VAR 
MesDataExd				: Datalogger_SENECA;                		
	
//INPUT Modbus
	FB_ModbusRead	          	: ARRAY[1..2] OF FB_ModbusRead; 	            // (NA) FB for Modbus Reading	
	MesBlock1_Temp				: ARRAY [1..8] OF WORD ; 
	
	AlarmModbusInput			: BOOL;
	AlarmID_ModbusInput			: UDINT;
END_VAR

METHOD M_AlarmManagement
//////////////////
// Generates object alarms and manages resets 
//////////////////

VAR 
	// Method local variables (reinitialized at each cycle) 
	FB_AlarmCodeManager		: FB_AlarmCodeManager;  
	Transfo_Synthesis		: INT;
END_VAR
	
// ALARM CODE //
	FB_AlarmCodeManager(
		bAlarm1				:= FALSE,														// 
		bAlarm2				:= FALSE,														// 
		bAlarm3				:= FALSE,														// 
		bAlarm4				:= FALSE,														//
		bAlarm5				:= FALSE,														//
		bAlarm6				:= FALSE,														//
		bAlarm7				:= FALSE,														//
		bAlarm8				:= FALSE,														//
		bAlarm9				:= FALSE,														//
		bAlarm10			:= FALSE,														//
		bAlarm11			:= FALSE, 														// 
		bAlarm12			:= FALSE, 														// 
		bAlarm13			:= FALSE, 														//                                          
		bAlarm14			:= FALSE,														//                                          
		bAlarm15			:= FALSE,														// 		
		wAlarmCode			=>MesDataExd.MesData.MesAlarmCode);										//
			
// WARNING CODE //
	FB_AlarmCodeManager(
		bAlarm1				:= AlarmModbusInput, 											// Error Modbus read of the datalogger data
		bAlarm2				:= FALSE, 														//
		bAlarm3				:= FALSE,														//
		bAlarm4				:= FALSE,														//
		bAlarm5				:= FALSE,														//
		bAlarm6				:= FALSE,														//
		bAlarm7				:= FALSE,														//
		bAlarm8				:= FALSE,														//
		bAlarm9				:= FALSE,														//
		bAlarm10			:= FALSE,														//
		bAlarm11			:= FALSE,														//
		bAlarm12			:= FALSE,														//
		bAlarm13			:= FALSE,														//
		bAlarm14			:= FALSE,														//
		bAlarm15			:= FALSE,														//
		wAlarmCode			=>MesDataExd.MesData.MesWarningCode);										//
		                                                        							
// EVENT CODE //                                                							                                                     							
	FB_AlarmCodeManager(                                        							
		bAlarm1				:= FALSE,						    							//  
		bAlarm2				:= FALSE, 														//  
		bAlarm3				:= FALSE,														//
		bAlarm4				:= FALSE,														//
		bAlarm5				:= FALSE,														//
		bAlarm6				:= FALSE,														//
		bAlarm7				:= FALSE,														//
		bAlarm8				:= FALSE,														//
		bAlarm9				:= FALSE,														//
		bAlarm10			:= FALSE,														//
		bAlarm11			:= FALSE,														//
		bAlarm12			:= FALSE,														//
		bAlarm13			:= FALSE,														//
		bAlarm14			:= FALSE,														//
		bAlarm15			:= FALSE,														//
		wAlarmCode			=>MesDataExd.MesData.MesEventCode);										//
		
MesDataExdMesDataExd		:= MesDataExd.MesData.
END_METHOD

METHOD M_CP

VAR 
	// Method local variables (reinitialized at each cycle) 
	
END_VAR

Trig_Cmd_Read(CLK:=IN_CmdToggleRead);

IF Trig_Cmd_Read.Q THEN
	IN_CmdToggleRead := FALSE;
	MesCP_Read := NOT MesCP_Read;
END_IF
END_METHOD

METHOD M_Execute : BOOL
VAR_INPUT
END_VAR
IF bInit THEN
	M_Init();
	bInit := FALSE;
ELSIF CmdInit_G THEN 
	bInit:= TRUE ;
END_IF

SUPER^.M_Execute() ;
END_METHOD

METHOD M_Init : BOOL
VAR_INPUT
END_VAR
END_METHOD


METHOD M_Read : BOOL
VAR_INPUT
END_VAR

VAR
	MW					: FB_MergeWordsToFloat;
END_VAR
// CP-Read / Write 

MesDataExd.MesData.MesCP_Read := MesCP_Read ; 
MesDataExd.MesData.MesCP_Write := MesCP_Write ;  

IF MesCP_Read  THEN	
// MODBUS Read	
	FB_ModbusRead[1]
		(
			nTCPPort		:= ParamTcpPort,
			ClockRead		:= MesCP_Read AND ClockRead, 
			Reset			:= CmdClearFault_G OR IN_CmdReset_L,
			sIPAddr			:= ParamIPAddress ,
			nUnitID			:= 1, 
			tTimeout		:= ParamWriteTimeout,
			nQuantity		:= 4, 
			nMBAddr			:= 40005, 
			cbLength		:= SIZEOF(MesBlock1_Temp), 
			pDestAddr		:= ADR(MesBlock1_Temp), 
			ModbusReadAlarm	=> AlarmModbusInput, 
			ErrorId			=> AlarmID_ModbusInput
		);
	
// Wind Data : Float AB CD	
	MW( WORD_STRONG:= MesBlock1_Temp[1  ],	WORD_WEAK := MesBlock1_Temp[2  ], VAR_OUT := MesDataExd.MesData.MesWindSp);		
	MW( WORD_STRONG:= MesBlock1_Temp[3  ],	WORD_WEAK := MesBlock1_Temp[4  ], VAR_OUT := MesDataExd.MesData.MesWindDir);
END_IF
END_METHOD

METHOD M_Write : BOOL
VAR
		
		
END_VAR
END_METHOD

END_FUNCTION_BLOCK

// ---- 01_Equipement_Library/GRID/FB_GRID_Base.TcPOU
FUNCTION_BLOCK FB_GRID_Base 
//////////////////
// Grid Operator interface. Base FB.
//////////////////
VAR_INPUT PERSISTENT
	// Parameters of the Object (instance specific) 
	
END_VAR

VAR_INPUT
	// I/O Inputs 
		MesConnectOrderIO			: BOOL ; 					// (NA) 
		MesDisconnectOrderIO 		: BOOL ; 					// (NA) 	
		
END_VAR

VAR_OUTPUT
	//Child objects
	
END_VAR
VAR
	//M_ALARMMANAGEMENT VARIABLES//                                                    								
//	MesDataExd				: GRID ;                   								
		
	//M_INIT VARIABLES //
		bInit						: BOOL:= TRUE ; 			// (NA) Initialize object parameters at first cycle 
		
	// M_EXECUTE VARIABLES //
	
   		MesCP_Read					: BOOL := TRUE;	(* Read function enable *)
		

                      	
END_VAR

METHOD M_AlarmManagement
//////////////////
// Digiware measurement tool alarm and warning management
/////////////////

VAR 
	
END_VAR
END_METHOD

METHOD M_CP

VAR 
	// Method local variables (reinitialized at each cycle) 
	
END_VAR
END_METHOD

METHOD M_Evaluate
//////////////////
//  Read Modbus Variable for PCS. 
/////////////////
VAR 
	// Method local variables (reinitialized at each cycle) 
	
END_VAR
END_METHOD

METHOD M_Execute
//////////////////
//  Method Calls 
/////////////////
VAR 
	// Method local variables (reinitialized at each cycle) 

END_VAR

// PERMANENT CONDITIONS //
	M_CP() ; 
	
// METHODS CALLS //
	IF bInit THEN
		M_Init() ; 
		bInit					:= FALSE ; 
	ELSIF CmdInit_G THEN 
		bInit:= TRUE ;
		
	END_IF

	M_Evaluate() ; 
	M_AlarmManagement();
END_METHOD

METHOD M_Init
VAR 

END_VAR
END_METHOD

END_FUNCTION_BLOCK

// ---- 01_Equipement_Library/GRID/FB_GRID_Enedis.TcPOU
FUNCTION_BLOCK FB_GRID_Enedis EXTENDS FB_GRID_Base
//////////////////
// Grid Operator interface. Base FB
//////////////////
VAR_INPUT PERSISTENT
	// Parameters of the Object (instance specific) 
		{attribute 'OPC.UA.DA' := '1'} 
		ParamRseAvailable						: BOOL:=TRUE;		(* (NA) GRID with RSE option*)
		{attribute 'OPC.UA.DA' := '1'} 
		ParamTaAvailable						: BOOL:=TRUE;		(* (NA) GRID with Teleaction option*)
		{attribute 'OPC.UA.DA' := '1'} 
		ParamP0Available						: BOOL:=TRUE; 		(* (NA) GRID with P regulation option*)
		{attribute 'OPC.UA.DA' := '1'} 
		ParamQ0Available						: BOOL:=TRUE; 		(* (NA) GRID with Q regulation option*)
		ParamTONFiltering						: TIME:=T#200MS; 	(* (ms) Minimum tempo filter before command validation (noise filtering)*)
		{attribute 'OPC.UA.DA' := '1'} 
		ParamPmaxPark							: REAL;				(* (kW) Contractual maximal power plant active power*)
		{attribute 'OPC.UA.DA' := '1'} 
		ParamQMax								: REAL;				(* (Kvar) Contractual maximal power plant reactive power*)
		{attribute 'OPC.UA.DA' := '1'} 
		ParamQMin								: REAL; 			(* (Kvar) Contractual maximal power plant reactive power*)
		{attribute 'OPC.UA.DA' := '1'} 
		ParamPMin								: REAL;				(* (kW)   Contractual minimal power plant active power*)
		
		MesDataExd								: GRID_Enedis;
END_VAR


VAR_INPUT
	// I/O Inputs 
		//FROM ENEDIS
		IN_CmdAutCpl_IO							: BOOL; 			//Coupling Authorization (Autorisation de couplage				)
		IN_CmdDisconnect_End_IO					: BOOL; 			//End of disconnect order(Fin de demande de decouplage         )
		IN_CmdDisconnect_IO						: BOOL;				//Disconnect order(Demande de decouplage                )
		IN_CmdRSEOn_IO							: BOOL;				//Start of RSE (Mise en RSE                          )
		IN_CmdRSEOff_IO							: BOOL;				//Stop of RSE (Mise Hors RSE                        )
		IN_CmdTAOn_IO							: BOOL; 			//Teleaction in service(Teleaction en service                )
		IN_CmdTAOff_IO							: BOOL; 			//Teleaction out of service (Teleaction Hors service              )
		IN_CmdStopPReg_IO						: BOOL;				//Desactivation of P0 regulation(Fin de passage a P0                  )
		IN_CmdStartPReg_IO						: BOOL;				//Activation of P0 regulation (Passage a P0                         )
		IN_CmdStopQReg_IO						: BOOL;				//Desactivation of Q0 regulation(Fin de passage a Q0                  )
		IN_CmdStartQreg_IO						: BOOL;				//Activation of Q0 regulation(Passage a Q0                         )
		IN_CmdEmergencyDisconnect_End_IO		: BOOL;				// End of Emergency disconnect order(Fin demande d'effacement d'urgence	)	
		IN_CmdEmergencyDisconnect_IO			: BOOL;				// Emergency disconnect order(Demande d'effacement d'urgence       )
		IN_CmdDisconnectFromTac_IO				: BOOL; 			// Teleaction disconnect(Decouplage par tac                   )
		IN_CmdTacInFault_IO						: BOOL; 			//Teleaction in fault(Défaut Tac							)
		IN_CmdSynchro_IO						: BOOL;				// Syncrhonization signal
		(* 4..20mA *)                                   			
		IN_MesP0Reg_IO							: INT; 				// (kW) Grid P0
		IN_MesQ0Reg_IO							: INT; 				// (Kvar) Grid Q0
		                                                			
		                                                			
		//FROM AKSES                                    			
		IN_CmdAutCpl_other						: BOOL; 			
		IN_CmdEmergencyDisconnect_other			: BOOL; 			
		IN_CmdEmergencyDisconnect_End_other		: BOOL; 			
		IN_CmdDisconnect_other					: BOOL; 			
		IN_CmdDisconnect_end_other				: BOOL; 			
		IN_CmdStartPReg_other					: BOOL; 			
		IN_CmdStartQReg_other					: BOOL; 			
		IN_CmdStopPReg_other					: BOOL; 			
		IN_CmdStopQReg_other					: BOOL; 			
		                                                			
		(*TC Relais Protection*)                        			
		IN_ConnectAuthorizationLost				: BOOL; 			// Tous les cas pour un Reset aut Couplage recu
		IN_Unavailable							: BOOL; 			// Disjoncteur général en Local, ou tous les départs en Local ou Bouton d'arret d'urgence 
		IN_PP_Connected							: BOOL; 			// Centrale Couplée si DG = Fermé et au moins 1 départ antenne en production et au moins un onduleur en Prod
                                                        			
END_VAR                                                 			
                                                        			
                                                        			
VAR_OUTPUT                                              			
		OUT_MesPPUnavailable_IO					: BOOL; 			// TS centrale indisponible
		OUT_MesPPConnected_IO					: BOOL; 			// Centrale couplée(1)/Centrale Découplée(0)
		OUT_MesPPDisconnected_IO				: BOOL; 			(*Centrale Découplée*)
		OUT_MesAutCpl_IO 						: BOOL; 			// Autorisation de couplage reçue(1)/Attente d'autorisation de couplage(0)
		OUT_MesAutCpl_end_IO 					: BOOL; 			(*Autorisation de couplage attente*)
		OUT_MesDisconnect_IO 					: BOOL; 			// Demande de découplage reçue(1)/Fin de demande de découplage(0)
		OUT_MesDisconnect_End_IO 				: BOOL; 			(*Demande de découplage attente*)
		OUT_MesEmergencyDisconnect_IO 			: BOOL; 			// Demande d effacement d'urgence reçue
		OUT_MesEmergencyDisconnect_End_IO 		: BOOL; 			(*Demande d effacement d'urgence attente*)		
		OUT_MesRSEON_IO							: BOOL; 			// Demande mise en RSE reçue
		OUT_MesRSEOff_IO						: BOOL; 			// Demande mise en RSE en attente
		OUT_MesTAOn_IO							: BOOL; 			// Demande mise en TeleAction reçue
		OUT_MesTAOff_IO							: BOOL; 			// Demande mise en TeleAction en attente
		OUT_MesStartPReg_IO						: BOOL; 			// Demande mise en regulation de P reçue
		OUT_MesStopPReg_IO						: BOOL; 			// Demande mise en regulation de P en attente
		OUT_MesStartQReg_IO						: BOOL; 			// Demande mise en regulation de Q reçue
		OUT_MesStopQReg_IO						: BOOL; 			// Demande mise en regulation de Q en attente	
END_VAR

VAR
		//TON
		TONConnectAuthorization					: TON;
		TONEmergencyDisconnect	               	: TON;
	    TONEmergencyDisconnect_end	            : TON;
	    TONDisconnect	                		: TON;
	    TONDisconnect_end                		: TON;
	    TONPRegOn				                : TON;
	    TONPRegOff				                : TON;
	    TONQregOn				                : TON;
	    TONQRegOff				                : TON;
	    TONRSEOn				                : TON;
	    TONRSEOff				                : TON;
	    TONTAOn					                : TON;
	    TONTAOff				                : TON;
				
END_VAR

METHOD M_AlarmManagement
//////////////////
// alarm and warning management
/////////////////

VAR 
	FB_AlarmCodeManager			: FB_AlarmCodeManager ; 
	
END_VAR
// ALARM CODE //
	FB_AlarmCodeManager(
		bAlarm1			:=MesDataExd.MesData.OUT_MesPPUnavailable, // Power plant is unavailable
		bAlarm2			:=FALSE, //
		bAlarm3			:=FALSE, //
		bAlarm4			:=FALSE, //
		bAlarm5			:=FALSE, //
		bAlarm6			:=FALSE, //
		bAlarm7			:=FALSE, //
		bAlarm8			:=FALSE, //
		bAlarm9			:=FALSE, //
		bAlarm10		:=FALSE, //
		bAlarm11		:=FALSE, //
		bAlarm12		:=FALSE, //
		bAlarm13		:=FALSE, //
		bAlarm14		:=FALSE, //
		bAlarm15		:=FALSE, //						 
		wAlarmCode		=>MesDataExd.MesData.MesAlarmCode);

// WARNING CODE //
	FB_AlarmCodeManager(		
		bAlarm1			:=IN_ConnectAuthorizationLost, 							//Loss of coupliong authorization
		bAlarm2			:=FALSE,													//			
		bAlarm3			:=MesDataExd.MesData.OUT_SetptP > ParamPmaxPark OR MesDataExd.MesData.OUT_SetptP <= 0 ,		// P Setpoint from grid outside of permitted range
		bAlarm4			:=MesDataExd.MesData.OUT_SetptQ > ParamQMax OR MesDataExd.MesData.OUT_SetptQ <= ParamQMin, 	// Q Setpoint from grid outside of permitted range
		bAlarm5			:=MesDataExd.MesData.OUT_MesPPConnected						, 	//Powerplant is connected  
		bAlarm6			:=NOT MesDataExd.MesData.OUT_MesPPConnected					, 	//Powerplant is disconnected
		bAlarm7			:=MesDataExd.OUT_CmdPReg							    , 	//Q regulation mode is active     
		bAlarm8			:=NOT MesDataExd.MesData.OUT_CmdAutCpl		    		, 	//Waiting for coupling authorization	
		bAlarm9			:=MesDataExd.MesData.OUT_CmdDisconnect				, 	//Disconnect order
		bAlarm10		:=MesDataExd.MesData.OUT_CmdEmergencyDisconnect 	        , 	//Emergency Disconnect order
		bAlarm11		:=MesDataExd.OUT_CmdPReg												, 	// P regulation mode is active
		bAlarm12		:=MesDataExd.OUT_Rse								    , 	// RSE mode active  
		bAlarm13		:=MesDataExd.OUT_TA 							, 	//Teleaction active
		bAlarm14		:=IN_CmdDisconnectFromTac_IO , 		// Disconnect order from TAC
		bAlarm15		:=IN_CmdTacInFault_IO , 			// TAC in Fault 
		wAlarmCode		=>MesDataExd.MesData.MesWarningCode);		

// EVENT CODE 1//
	FB_AlarmCodeManager(
		bAlarm1			:=FALSE , // 
		bAlarm2			:=NOT MesDataExd.OUT_CmdPReg							    , 	//P regulation mode is inactive
		bAlarm3			:=MesDataExd.MesData.OUT_CmdAutCpl					, 	//Coupling authorization
		bAlarm4			:=FALSE ,//
		bAlarm5			:=IN_CmdSynchro_IO			    						, 	// Synchronization signal 
		bAlarm6			:=NOT MesDataExd.MesData.OUT_CmdDisconnect			, 	//End of disconnect order 
		bAlarm7			:=MesDataExd.MesData.OUT_CmdDisconnect				, 	//Disconnect order
		bAlarm8			:=NOT MesDataExd.MesData.OUT_CmdEmergencyDisconnect					, 	//End of Emergency Disconnect order
		bAlarm9			:=MesDataExd.MesData.OUT_CmdEmergencyDisconnect 	        , 	//Emergency Disconnect order
		bAlarm10		:=MesDataExd.OUT_CmdPReg												, 	// P regulation mode is active
		bAlarm11		:=NOT MesDataExd.OUT_CmdPReg												, 	//P regulation mode is inactive
		bAlarm12		:=MesDataExd.OUT_Rse								    , 	// RSE mode active    
		bAlarm13		:=NOT MesDataExd.OUT_Rse							    , 	//RSE mode inactive  
		bAlarm14		:=MesDataExd.OUT_TA 							, 	//Teleaction active
		bAlarm15		:=NOT MesDataExd.OUT_TA							, 	//Teleaction inactive
		wAlarmCode		=>MesDataExd.MesData.MesEventCode);   
                          	
// EVENT CODE 2 //		                                              	
	FB_AlarmCodeManager(                                              	
		bAlarm1			:=IN_CmdAutCpl_IO , 							// Autorisation de couplage du DEIE
		bAlarm2			:=IN_CmdDisconnect_End_IO,						// Fin de demande de découplage du DEIE
		bAlarm3			:=IN_CmdDisconnect_IO		   , 				// Demande de decouplage du DEIE
		bAlarm4			:= IN_CmdEmergencyDisconnect_End_IO	   	, 		// Emergency disconnect
		bAlarm5			:=IN_CmdAutCpl_other, 							// Autorisation de couplage du DEIE de la HMI
		bAlarm6			:=IN_CmdDisconnect_other		 , 				// Demande de decouplage du DEIE de la HMI
		bAlarm7			:=IN_CmdDisconnect_end_other,	 				// Demande de decouplage par TAC de la HMI
		bAlarm8			:=FALSE	, 										// 
		bAlarm9			:=IN_Unavailable, 								// Centrale indisponible dans le code
		bAlarm10		:=FALSE, 	//
		bAlarm11		:=FALSE	, 	//
		bAlarm12		:=FALSE, 	//
		bAlarm13		:=FALSE, 	//       
		bAlarm14		:=FALSE, 	//
		bAlarm15		:=FALSE	,//
		wAlarmCode		=>MesDataExd.MesData.MesEventCode2);
END_METHOD

METHOD M_CP
//////////////////
//  Emulator
/////////////////

VAR 
	// Method local variables (reinitialized at each cycle) 
	
END_VAR
END_METHOD

METHOD M_Evaluate
//////////////////
//  Evaluate grid variables 
/////////////////
VAR 
	// Method local variables (reinitialized at each cycle) 
	WatchDog	: BOOL;
END_VAR
WatchDog		:= TRUE;

//Filtering Input
	TONConnectAuthorization		(IN:=IN_CmdAutCpl_IO,PT:=ParamTONFiltering);
	TONEmergencyDisconnect		(IN:=IN_CmdEmergencyDisconnect_IO,PT:=ParamTONFiltering);	
	TONEmergencyDisconnect_end	(IN:=IN_CmdEmergencyDisconnect_End_IO,PT:=ParamTONFiltering);	
	TONDisconnect				(IN:=IN_CmdDisconnect_IO,PT:=ParamTONFiltering);	
	TONDisconnect_end			(IN:=IN_CmdDisconnect_End_IO,PT:=ParamTONFiltering);
	TONPRegOn				(IN:=IN_CmdStartPReg_IO,PT:=ParamTONFiltering);			
	TONPRegOff				(IN:=IN_CmdStopPReg_IO,PT:=ParamTONFiltering);				
	TONQregOn				(IN:=IN_CmdStartQreg_IO,PT:=ParamTONFiltering);				
	TONQRegOff				(IN:=IN_CmdStopQReg_IO,PT:=ParamTONFiltering);				
	TONRSEOn				(IN:=IN_CmdRSEOn_IO,PT:=ParamTONFiltering);				
	TONRSEOff				(IN:=IN_CmdRSEOff_IO,PT:=ParamTONFiltering);				
	TONTAOn					(IN:=IN_CmdTAOn_IO,PT:=ParamTONFiltering);					
	TONTAOff				(IN:=IN_CmdTAOff_IO,PT:=ParamTONFiltering);		

//Converting P0 & Q0
	IF ParamP0Available THEN
		//OUT_P0 :=  (MesP0RegIO/ 32767.0) * REAL_TO_INT(ParamPmaxPark);
	MesDataExd.MesData.OUT_SetptP :=  (IN_MesP0Reg_IO/ 32767.0) * ABS(ParamPMin - ParamPmaxPark) + (ParamPMin);
	END_IF
	IF ParamQ0Available THEN
	MesDataExd.MesData.OUT_SetptQ := ( IN_MesQ0Reg_IO / 32767.0) * ABS(ParamQMin - ParamQMax) + (ParamQMin);
	END_IF	
//Logical Equation
	(*PLCUnavailable Si Watchdog n'est pas mis a jour a chaque temps de cycle Ou que la centrale est en Local *)
	MesDataExd.MesData.OUT_MesPPUnavailable := NOT WatchDog OR IN_Unavailable;
	
	(*Centrale Couplée *)
	MesDataExd.MesData.OUT_MesPPConnected := IN_PP_Connected;
	
	(*Autorisation de couplage*)
		IF TONConnectAuthorization.Q OR IN_CmdAutCpl_other THEN
		MesDataExd.MesData.OUT_CmdAutCpl := 1 ;
		END_IF
		
	(*Défaut GTE > 50s : Reset Aut Couplage recus*)
	(*Défaut C13_100 : Reset Aut Couplage recus*)
		IF IN_ConnectAuthorizationLost THEN  //IN_Long_GTE_Fault OR IN_C13_100_Fault OR IN_UnknownFault OR IN_3GTE_Fault THEN
		MesDataExd.MesData.OUT_CmdAutCpl  := FALSE ;
		END_IF
	
	(* RESEAU 6 ET 7 - DEMANDE DE DECOUPLAGE*)
		IF TONDisconnect.Q OR IN_CmdDisconnect_other THEN
			MesDataExd.MesData.OUT_CmdDisconnect := 1 ;
		END_IF
	
		IF TONDisconnect_end.Q OR IN_CmdDisconnect_end_other THEN
		MesDataExd.MesData.OUT_CmdDisconnect := 0 ;
		END_IF

	(* RESEAU 8 ET 9 - DEMANDE D’EFFACEMENT D’URGENCE*)
		IF TONEmergencyDisconnect.Q OR  IN_CmdEmergencyDisconnect_other THEN
		MesDataExd.MesData.OUT_CmdEmergencyDisconnect := 1 ;
		END_IF
	
		IF TONEmergencyDisconnect_end.Q OR IN_CmdEmergencyDisconnect_End_other THEN
		MesDataExd.MesData.OUT_CmdEmergencyDisconnect := 0 ;
		END_IF
	(* RESEAU 10 ET 11 - PASSAGE A P0*)
		IF TONPRegOn.Q OR IN_CmdStartPReg_other THEN
		MesDataExd.OUT_CmdPReg := 1 ;
		END_IF
		
		IF TONPRegOff.Q OR IN_CmdStopPReg_other THEN
		MesDataExd.OUT_CmdPReg := 0 ;
		END_IF
		
	(* RESEAU 12 ET 13 - PASSAGE A Q0*)
		IF TONQregOn.Q OR IN_CmdStartQReg_other THEN
		MesDataExd.OUT_CmdQReg := 1 ;
		END_IF
		
		IF TONQregOff.Q OR IN_CmdStopQReg_other THEN
		MesDataExd.OUT_CmdQReg := 0 ;
		END_IF

				
	(* RSE*)
		IF TONRSEOn.Q  THEN
		MesDataExd.OUT_Rse := 1 ;
		ELSIF TONRSEOff.Q THEN
		MesDataExd.OUT_Rse := 0 ;
		END_IF
		
	(* TA*)
		IF TONTAOn.Q  THEN
		MesDataExd.OUT_TA := 1 ;
		ELSIF TONTAOff.Q THEN
		MesDataExd.OUT_TA := 0 ;
		END_IF
		
	
// Update Outputs IO to GRID 
OUT_MesPPUnavailable_IO				:= MesDataExd.MesData.OUT_MesPPUnavailable ; 			
OUT_MesPPConnected_IO				:= MesDataExd.MesData.OUT_MesPPConnected ; 	
OUT_MesPPDisconnected_IO			:= NOT MesDataExd.MesData.OUT_MesPPConnected ; 
OUT_MesAutCpl_IO 					:= MesDataExd.MesData.OUT_CmdAutCpl ; 			
OUT_MesAutCpl_end_IO 				:= NOT MesDataExd.MesData.OUT_CmdAutCpl ; 		
OUT_MesDisconnect_IO 				:= MesDataExd.MesData.OUT_CmdDisconnect ; 		
OUT_MesDisconnect_End_IO 			:= NOT MesDataExd.MesData.OUT_CmdDisconnect ; 		
OUT_MesEmergencyDisconnect_IO 		:= MesDataExd.MesData.OUT_CmdEmergencyDisconnect ; 		
OUT_MesEmergencyDisconnect_End_IO 	:= NOT MesDataExd.MesData.OUT_CmdEmergencyDisconnect ; 		

OUT_MesRSEON_IO						:= MesDataExd.OUT_Rse ;
OUT_MesRSEOff_IO					:= NOT MesDataExd.OUT_Rse ;
OUT_MesTAOn_IO						:= MesDataExd.OUT_TA ; 
OUT_MesTAOff_IO						:= NOT MesDataExd.OUT_TA ; 

OUT_MesStartPReg_IO	 := MesDataExd.OUT_CmdPReg ; 
OUT_MesStopPReg_IO	 := NOT MesDataExd.OUT_CmdPReg ; 
OUT_MesStartQReg_IO	 := MesDataExd.OUT_CmdQReg ; 
OUT_MesStopQReg_IO	 := NOT MesDataExd.OUT_CmdQReg ;
END_METHOD

METHOD M_Execute
//////////////////
//  Method Calls 
/////////////////
VAR 
	// Method local variables (reinitialized at each cycle) 
	
END_VAR
// PERMANENT CONDITIONS //
	M_CP() ; 
	
// METHODS CALLS //
	IF bInit THEN
		M_Init() ; 
		bInit:= FALSE ; 
	ELSIF CmdInit_G THEN 
		bInit:= TRUE ;
	END_IF

	M_Evaluate() ; 
	M_AlarmManagement();
END_METHOD

METHOD M_Init
VAR 

END_VAR
// Au démarrage du code , on maintient en mémoire l'autorization de couplage ssi la centrale est connectée. 
IF NOT A1_SUBMV.A1_MainMVCB.MesDataExd.MesData.MesClosed THEN // La centrale n'est pas connectée
	MesDataExd.MesData.OUT_CmdAutCpl := FALSE ;
	MesDataExd.OUT_CmdPReg := FALSE;
	MesDataExd.OUT_CmdQReg := FALSE;

END_IF
END_METHOD

END_FUNCTION_BLOCK

// ---- 01_Equipement_Library/GRID/FB_GRID_MADI.TcPOU
FUNCTION_BLOCK FB_GRID_MADI EXTENDS FB_GRID_Base
//////////////////
// Grid Operator interface . Base FB
//////////////////
VAR_INPUT PERSISTENT
	// Parameters of the Object (instance specific) 

		ParamTONFiltering						: TIME:=T#500MS; 	(* Filtre tempo minimum avant validation de la commande (Filtrage du bruit)	*)
		ParamTONPulse							: TIME:=T#1S; 		(* Tempo to transform command to impulse .                                  *)
		{attribute 'OPC.UA.DA' := '1'}                                                                                                       
		ParamPmaxPark							: REAL;				(* Puissance max du park (Kw)                                               *)
		{attribute 'OPC.UA.DA' := '1'}                              
		ParamPminPark							: REAL ; 			(* puissance minimal du park                                                *)
		{attribute 'OPC.UA.DA' := '1'}                              
		ParamEmax								: REAL ; 			(* Maximal Contractual Energy .                                             *)
		                                                            
		ParamTempoComAlarm			: TIME 		:= T#10S;			(* Time before communication alarm	                                        *)
END_VAR


VAR_INPUT
	// I/O Inputs 
		//FROM AKSES
		IN_CmdAut_Cpl_other				: BOOL;
		IN_CmdDisconnect_other			: BOOL;	
		//IN_CmdConnect_other			: BOOL;	
		IN_CmdSoutirage_other			: BOOL;	
		IN_CmdInjection_other			: BOOL;			
		IN_CmdTest_other				: BOOL;	
		IN_CmdManualMode_other			: BOOL;
		IN_CmdManualModeOff_other		: BOOL;
	    IN_CmdToggleRead				: BOOL;	
		IN_ConnectAuthorizationLost		: BOOL; 

END_VAR 
VAR_OUTPUT
	//Child objects 17 OUtput
END_VAR

VAR PERSISTENT 
	MesDataExd				: GRID_MADI ; 
END_VAR

VAR
	//M_ALARMMANAGEMENT VARIABLES//                                                    								
		TON_ComAlarm							: TON;
		RS_ChargingAlarm						: RS;
	//M_EVALUATE VARIABLES//					
		//TON                       			
		TONConnectAuthorization					: TON;
		TONDisconnectOrder	        			: TON;
	    TONSoutirage	            			: TON;
	    TONTest	                				: TON;
	    TONModeManu				    			: TON;
		TONModeManuOff							: TON;
		TOF_ToS									: TOF;
                                                
                                                
		TONConnectAuthorizationPulse			: TON;
		TONDisconnectOrderPulse               	: TON;
	    TONModeManuPulse				        : TON;
		
		CheckCommand							: ARRAY[1..5] OF  FB_CheckCommand ;
		TON_CheckCommand						: ARRAY[1..5] OF TON ;
		
		OUT_MesEconnected						: REAL;// To be used for HMI only
		OUT_MesEmaxconnected					: REAL;
		OUT_MesIECServerFault					: BOOL;		
		
		RS_Soutirage_other						: RS;
		
	//M_Evaluate
		SetptP_old								: REAL;
		ParamPmax_old							: REAL ;
		ParamPmin_old							: REAL;		
                                        		
	// IEC 104                          		
	 	MesDataIEC								: IEC104;
		AODB 									: ARRAY[0..GVL_Cst.CstNbAOEntries] OF ST_IEC870_5_101AODBEntry ;
		memory 			AT%MB0					: ARRAY[0..79] OF BYTE;
		FB_IEC									: FB_IEC104ServerAkuo;(* Controlled station function block instance *)

	
	//M_INIT VARIABLES //
	//	bInit									: BOOL:= TRUE;	
		initError								: UDINT;
		bBoot									: BOOL := TRUE ; // Boolean that indicates a restart of the PLC .
	// M_EXECUTE VARIABLES //
        Trig_Cmd_Read							: R_TRIG;                                                                                        
		
		   		                    		
                     
				
END_VAR

METHOD M_AlarmManagement
//////////////////
// alarm and warning management
/////////////////

VAR 
	FB_AlarmCodeManager			: FB_AlarmCodeManager ; 
	

END_VAR
	TON_ComAlarm	(IN:= NOT( FB_IEC.eDTState =1 ) , PT:= ParamTempoComAlarm, 	Q=> MesDataExd.MesData.MesAlarmCom) ;	

	RS_ChargingAlarm(SET:= MesDataIEC.OUT_MesCharging , RESET1:= MesDataIEC.OUT_MesDischarging ) ; 
	
// ALARM CODE //
	FB_AlarmCodeManager(
		bAlarm1			:=MesDataIEC.IN_SetptP >MesDataIEC.IN_ParamPmax OR MesDataIEC.IN_SetptP < MesDataIEC.IN_ParamPmin, 	// Setpoint received outside of limits 
		bAlarm2			:=MesDataIEC.IN_Cmddouble.0 = MesDataIEC.IN_Cmddouble.1 , 												// Uncohetent not defined signal 
		bAlarm3			:=MesDataIEC.IN_Cmddouble.2 = MesDataIEC.IN_Cmddouble.3, 												// Uncoherent Start signal 
		bAlarm4			:=MesDataIEC.IN_Cmddouble.4 = MesDataIEC.IN_Cmddouble.5, 												// Uncoherent test signal
		bAlarm5			:=FALSE, 																								//
		bAlarm6			:=FALSE,                                                                                                //
		bAlarm7			:=FALSE,                                                                                                //
		bAlarm8			:=FALSE,                                                                                                //
		bAlarm9			:=FALSE, 																								//
		bAlarm10		:=FALSE,                                                                                                //
		bAlarm11		:=FALSE,                                                                                                //
		bAlarm12		:=FALSE,                                                                                                //
		bAlarm13		:=FALSE, 																								//
		bAlarm14		:=NOT MesCP_Read,																				// IEC 104 Disabled.  
		bAlarm15		:= MesDataExd.MesData.MesAlarmCom, 						 															// Communication alarm with IEC 104 #COM
		wAlarmCode		=>MesDataExd.MesData.MesAlarmCode);

// WARNING CODE //
	FB_AlarmCodeManager(		
		bAlarm1			:=RS_ChargingAlarm.Q1 , 														//Monitoring direction : PP is charging
		bAlarm2			:=NOT RS_ChargingAlarm.Q1, 														//Monitoring direction : PP is discharging
		bAlarm3			:= MesDataIEC.OUT_MesEs, 														//Monitoring direction : Emergency stop     
		bAlarm4			:= MesDataIEC.OUT_MesLocal, 														//Monitoring direction : Local Mode
		bAlarm5			:= MesDataIEC.OUT_MesModeAuto_on, 												//Monitoring direction : Frequency regulation in progress
		bAlarm6			:= MesDataIEC.OUT_MesModeManuel_on, 												//Monitoring direction : Manual Mode is active
		bAlarm7			:= MesDataIEC.OUT_MesToS, 														//Monitoring direction : Techician on site
		bAlarm8			:= MesDataIEC.MesCentrale_Cpl, 													//Monitoring direction : PP is connected to the grid
		bAlarm9			:= MesDataIEC.MesCentrale_indispo, 												//Monitoring direction : PP is unavailable
		bAlarm10		:= MesDataIEC.MesSoutirage_on, 														//Monitoring direction : PP is started
		bAlarm11		:= MesDataIEC.OUT_MesIECServerFault, 											//Monitoring direction : IEC server fault   
		bAlarm12		:= MesDataIEC.OUT_MesFaultTeleCmd, 												//Monitoring direction : TC server fault
		bAlarm13		:= MesDataIEC.OUT_MesFaultTeleSgnl, 												//Monitoring direction : TS server fault             
		bAlarm14		:= MesDataIEC.OUT_MesFaultTeleMes, 												//Monitoring direction : TM server fault               
		bAlarm15		:= MesDataIEC.OUT_MesIncident       ,       										//Monitoring direction : Incident       
		wAlarmCode		=>MesDataExd.MesData.MesWarningCode);		

// EVENT CODE 1//

	FB_AlarmCodeManager(
		bAlarm1			:= MesDataIEC.IN_CmdAut_Cpl	, 					// Control direction : Coupling autorization request
		bAlarm2			:=FALSE	, 							            //
		bAlarm3			:= MesDataIEC.IN_CmdModeManuel	, 	            // Control direction : Manual Mode activation request 
		bAlarm4			:= MesDataIEC.IN_CmdDisconnect    , 	            // Control direction : PP disconnection request 
		bAlarm5			:= MesDataIEC.CmdSoutirage    , 	                    // Control direction : PP soutirage request  
		bAlarm6			:=FALSE, 	                                    //
		bAlarm7			:=FALSE, 	                                    //
		bAlarm8			:=FALSE, 	                                    //
		bAlarm9			:=FALSE   , 	                                //
		bAlarm10		:=FALSE, 	                                    //
		bAlarm11		:=FALSE, 	                                    //
		bAlarm12		:=FALSE   , 	                                //
		bAlarm13		:=FALSE   , 	                                //
		bAlarm14		:=FALSE, 	                                    //
		bAlarm15		:=FALSE, 	                                    //
		wAlarmCode		=>MesDataExd.MesData.MesEventCode);
END_METHOD

METHOD M_CP
VAR 

END_VAR
Trig_Cmd_Read(CLK:=IN_CmdToggleRead);
	
IF Trig_Cmd_Read.Q THEN
	//IN_CmdToggleRead := FALSE;
	MesCP_Read := NOT MesCP_Read;
END_IF
END_METHOD

METHOD M_Evaluate
//////////////////
//  Read Modbus Variable for PCS . 
/////////////////
VAR 
	// Method local variables (reinitialized at each cycle) 
	KK: INT;
	CalTos: BOOL;
	CalEs: BOOL;

	CalComEss: BOOL;



	

END_VAR
	// Update values to be sent through IEC 104 . 

	//MesDataIEC.MesStart_on := A1_PP.MesDataExd.MesData.MesState.2 ; 		// Ecrit par le protocole comme un acquittement
	//MesDataIEC.MesComTest_on := ; 								// ecrit par le protocole comme un acquittement .
	
MesDataIEC.MesCentrale_Cpl :=  A1_PP.MesData.MesState.2  ;									
MesDataIEC.MesCentrale_indispo := A1_PP.MesData.MesPP_Unavailable ; // Alarmes feu, arret urgence, mode local , UPS en decharge , Puissance dispo trop faible , 
MesDataIEC.MesDJOpen  :=  A1_SUBMV.A1_MainMVCB.MesDataExd.MesData.MesOpened; // DJ open
	
	
	
(*.MesDataIEC.OUT_MesDouble.0 := NOT MesDataIEC.MesStart_on ; 
.MesDataIEC.OUT_MesDouble.1 := MesDataIEC.MesStart_on ; *)
(*.MesDataIEC.OUT_MesDouble.2 := MesDataIEC.MesComTest_on ; 
.MesDataIEC.OUT_MesDouble.3 := NOT MesDataIEC.MesComTest_on ; *) 
MesDataIEC.OUT_MesDouble.4 := MesDataIEC.MesCentrale_Cpl ; 
MesDataIEC.OUT_MesDouble.5 := NOT MesDataIEC.MesCentrale_Cpl ;
MesDataIEC.OUT_MesDouble.6 := MesDataIEC.MesCentrale_indispo ; 
MesDataIEC.OUT_MesDouble.7 := NOT MesDataIEC.MesCentrale_indispo ;

MesDataIEC.OUT_MesDouble.0 := NOT MesDataIEC.MesDJOpen ; 
MesDataIEC.OUT_MesDouble.1 := MesDataIEC.MesDJOpen ; 	
	
	(*
	CalEs	:= FALSE ;
	CalTos	:= FALSE ;
	CalComEss := FALSE;
	
	FOR KK:= 1 TO CstNbEss DO 
		CalTos := CalTos OR AX_ESS[KK].A1_ToS.MesDataExd.MesData.MesAlarmState OR AX_ESS[KK].A1_DS_Bat.MesDataExd.MesData.MesAlarmState OR AX_ESS[KK].A1_Ds_Pcs.MesDataExd.MesData.MesAlarmState ;
		CalEs	:= CalEs OR AX_ESS[KK].A1_ES.MesDataExd.MesData.MesAlarmState ;
		CalComEss := CalComESS OR AX_ESS[KK].AX_Bat[1].MesDataExd.MesData.MesAlarmCom OR AX_ESS[KK].AX_Bat[1].MesDataExd.MesData.MesAlarmCom ;
	END_FOR
	
.MesDataIEC.OUT_MesLocal			:= A1_PP.ParamLocalMode ; 
.MesDataIEC.OUT_MesModeManuel_on := A1_PP.MesDataExd.MesData.CalManualMode  ;
.MesDataIEC.OUT_MesModeAuto_on	:= A1_PP.MesDataExd.MesData.CalFreqMode  ;
.MesDataIEC.OUT_MesCharging		:= A1_PP.MesDataExd.MesData.MesPbat < - A1_SUBMV.A1_PM_Aux.MesDataExd.MesData.MesP - 500 ;   // Charging more than the auxiliaries  ( keep some margin  ). 
.MesDataIEC.OUT_MesDischarging	:= A1_PP.MesDataExd.MesData.MesPbat > 500 ;
.MesDataIEC.OUT_MesEs			:= A1_SUBMV.A1_TOR_Es.MesDataExd.MesData.MesAlarmState OR CalEs ; 
	TOF_ToS(IN:= A1_SUBMV.A1_DS_LV.MesDataExd.MesData.MesAlarmState OR 	A1_SUBMV.A1_TOR_DsHT.MesDataExd.MesData.MesAlarmState OR CalTos , PT:= T#1H , Q =>MesDataIEC.OUT_MesToS	)  ; 	
.MesDataIEC.OUT_MesIncident		:=  (*A1_PP.MesDataExd.MesData.MesAlarmCode.0 OR*) A1_SUBMV.MesDataExd.MesData.MesAlarmCode.0 ; // Alarm on the PP or SUB_MV . 	
.MesDataIEC.OUT_MesFaultTeleMes	:= A1_SUBMV. AX_PM[1].MesDataExd.MesData.MesAlarmCom AND A1_SUBMV.AX_PM[2].MesDataExd.MesData.MesAlarmCom OR CalComEss; // Si defaut de com sur un des signaux de la telemesure . 	
.MesDataIEC.OUT_MesFaultTeleCmd	:= CheckCommand[1].bWarning OR CheckCommand[2].bWarning OR CheckCommand[3].bWarning OR CheckCommand[4].bWarning OR CheckCommand[5].bWarning  ; // Si defaut d	
	/.MesDataIEC.OUT_MesFaultTeleSgnl	:=   ; // Si defaut d ecriture modbus des setpoint de P . 
	OUT_MesIECServerFault				:= SEL(CstPLCBackup ,NOT MAIN.OUT_CalRunningPLC_IO  ,MAIN.OUT_CalRunningPLC_IO ) ; // NOT MesCP_Read  ; // Define nwhich PA is active ( False  = PA 1  , else PA 2 )  
.MesDataIEC.OUT_MesIECServerFault	:= OUT_MesIECServerFault ;


	OUT_MesEconnected					:= A1_PP.MesDataExd.MesData.OUT_Econnected / 1000 ;	
.MesDataIEC.OUT_MesEconnected 		:= OUT_MesEconnected ;
	OUT_MesEmaxconnected 				:= A1_PP.MesDataExd.MesData.OUT_Enomconnected / 1000 ;			// MWh . Capacité maximale connectée ( taking account 12MWh max , and soc security .  
.MesDataIEC.OUT_MesEmaxconnected 	:= OUT_MesEmaxconnected; 
	
.MesDataIEC.OUT_MesP 			:= 	 A1_PP.MesDataExd.MesData.MesPbat /1000 ;		// MW
.MesDataIEC.OUT_MesQ 			:= 	 A1_PP.MesDataExd.MesData.MesQbat/1000 ;	// MVAr
.MesDataIEC.OUT_MesU_HTA 		:=	 A1_PP.MesDataExd.MesData.MesU/1000;		// kV
.MesDataIEC.OUT_MesFreq 			:= 	 A1_SUBMV.MesDataExd.MesData.MesFreq;		// Hz
.MesDataIEC.OUT_MesPdispo_inj 	:=  A1_PP.MesDataExd.MesData.OUT_SetptPmax  /1000 ; // MW
.MesDataIEC.OUT_MesPdispo_abs 	:=   A1_PP.MesDataExd.MesData.OUT_SetptPmin /1000 ; // MW 
*)
	// TREAT COMMANDS 
	// FAIRE DES IMPULSIONS SUR LES COMMANDES . 

	// Double point commands. 
MesDataIEC.CmdSoutirage := MesDataIEC.IN_Cmddouble.3 ;
MesDataIEC.CmdTest := MesDataIEC.IN_Cmddouble.4 ; 
	
	//Filtering Input
		TONConnectAuthorization	(IN:= MesDataIEC.IN_CmdAut_Cpl,PT:=ParamTONFiltering);
		TONDisconnectOrder		(IN:= MesDataIEC.IN_CmdDisconnect,PT:=ParamTONFiltering);		
		TONSoutirage	(IN:= MesDataIEC.CmdSoutirage,PT:=ParamTONFiltering);	
		TONTest	(IN:= MesDataIEC.CmdTest,PT:=ParamTONFiltering);	
		TONModeManu			(IN:= MesDataIEC.IN_CmdModeManuel,PT:=ParamTONFiltering);
		TONModeManuOff			(IN:= MesDataIEC.IN_CmdModeManuelOff,PT:=ParamTONFiltering);			



	// Impulsions
		TONConnectAuthorizationPulse	(IN:=TONConnectAuthorization.Q,PT:=ParamTONPulse);
		TONDisconnectOrderPulse		(IN:=TONDisconnectOrder.Q	,PT:=ParamTONPulse);		
		TONModeManuPulse		(IN:=TONModeManu.Q,PT:=ParamTONPulse);	

	RS_Soutirage_other(SET:=IN_CmdSoutirage_other , RESET1:=IN_CmdInjection_other (*OR MesDataExd.MesData.OUT_CmdDisconnect*)) ; 
	
	(*Autorisation de couplage*)
	IF TONConnectAuthorization.Q AND NOT A1_PP.ParamLocalMode OR A1_PP.ParamLocalMode AND IN_CmdAut_Cpl_other THEN
	MesDataExd.MesData.OUT_CmdAutCpl := TRUE ;
	MesDataExd.MesData.OUT_CmdDisconnect := FALSE ; 
		IF TONConnectAuthorizationPulse.Q THEN 
		MesDataIEC.IN_CmdAut_Cpl := FALSE ; // Reinitialize to false the input to get an impulse. 
		END_IF
	END_IF
	IF IN_ConnectAuthorizationLost THEN  //IN_Long_GTE_Fault OR IN_C13_100_Fault OR IN_UnknownFault OR IN_3GTE_Fault  OR CmdDecouplage 
	MesDataExd.MesData.OUT_CmdAutCpl := FALSE ;
	END_IF
	
	IF TONDisconnectOrder.Q AND NOT A1_PP.ParamLocalMode OR A1_PP.ParamLocalMode AND IN_CmdDisconnect_other THEN 
	MesDataExd.MesData.OUT_CmdDisconnect := TRUE ; 
	MesDataExd.MesData.OUT_CmdAutCpl := FALSE ;
		IF TONDisconnectOrderPulse.Q THEN 
		MesDataIEC.IN_CmdDisconnect := FALSE ; // Reinitialize to false the input to get an impulse.
		END_IF
	END_IF
	//  MesDataExd.MesData.OUT_CmdAut_Cpl := TONConnectAuthorization.Q OR A1_PP.ParamLocalMode AND IN_CmdAut_Cpl_other ; 	// Impulse // ADD LOCAL ONLY 

	IF 	TONModeManuPulse.Q 	AND NOT A1_PP.ParamLocalMode THEN 
	MesDataIEC.IN_CmdModeManuel := FALSE ; // Reinitialize to false the input to get an impulse.
	END_IF
	
	//  MesDataExd.MesData.OUT_CmdDisconnect := TONDisconnectOrder.Q 	OR A1_PP.ParamLocalMode AND IN_CmdDisconnect_other		; 
(*
MesDataExd.MesData.OUT_CmdModeManuel := TONModeManu.Q 	AND NOT A1_PP.ParamLocalMode		OR A1_PP.ParamLocalMode AND IN_CmdManualMode_other	; 	// Impulse
MesDataExd.MesData.OUT_CmdModeManuelOff := TONModeManuOff.Q 	AND NOT A1_PP.ParamLocalMode		OR A1_PP.ParamLocalMode AND IN_CmdManualModeOff_other	; 	// Impulse
MesDataExd.MesData.OUT_CmdSoutirage := (TONSoutirage.Q 		AND NOT A1_PP.ParamLocalMode 		OR  A1_PP.ParamLocalMode AND	RS_Soutirage_other.Q1) AND NOT MesDataExd.MesData.OUT_CmdDisconnect ;	// True / False . 
MesDataExd.MesData.OUT_CmdTest := TONTest.Q 		AND NOT A1_PP.ParamLocalMode			OR A1_PP.ParamLocalMode AND IN_CmdTest_other		; 
	*)
	// Write value only on change . 
	IF MesDataIEC.IN_SetptP <> SetptP_old THEN 
	MesDataExd.MesData.OUT_SetptP 				:= MesDataIEC.IN_SetptP *1000  ;  
		SetptP_old := MesDataIEC.IN_SetptP ; 
	END_IF

(*	IF MesDataIEC.IN_ParamPmax <> ParamPmax_old THEN 
	MesDataExd.MesData.OUT_ParamPmax			:=	MIN(MesDataIEC.IN_ParamPmax*1000 , ParamPmaxPark)  ;  
		ParamPmax_old := MesDataIEC.IN_ParamPmax   ; 
	END_IF	
	IF MesDataIEC.IN_ParamPmin <> ParamPmin_old THEN 
	MesDataExd.MesData.OUT_ParamPmin				:=	MAX( MesDataIEC.IN_ParamPmin*1000, ParamPminPark)   ;  
		ParamPmin_old := MesDataIEC.IN_ParamPmin ; 
	END_IF	
*)

	// Detect if command is not applied  
	// Start 
	TON_CheckCommand[1](IN:= CheckCommand[1].bWarning , PT:= T#2S ) ; 
	CheckCommand[1](
		bCmd		:= MesDataExd.MesData.OUT_CmdAutCpl  ,
		bMes		:= A1_PP.MesData.MesState.2 , 		// Compare with the modbus feedback on equipement . 
		bReset		:= TON_CheckCommand[1].Q,		// Reset after 2 se
		bImpulsion	:= TRUE , 
		T			:= T#120S ) ;
(*		
	// Stop Mode 
	TON_CheckCommand[2](IN:= CheckCommand[2].bWarning , PT:= T#2S ) ; 
	CheckCommand[2](
		bCmd		:=  NOT MesDataExd.MesData.OUT_CmdSoutirage ,
		bMes		:= A1_PP.MesDataExd.MesData.MesState.0 , 		// Compare with the modbus feedback on equipement . 
		bReset		:=TON_CheckCommand[2].Q ,
		bImpulsion	:= TRUE , 
		T			:= T#5S ) ;	
	*)
	// Disconnect 
	TON_CheckCommand[3](IN:= CheckCommand[3].bWarning , PT:= T#2S ) ; 
	CheckCommand[3](
		bCmd		:= MesDataExd.MesData.OUT_CmdDisconnect,
		bMes		:= A1_PP.MesData.MesState.0 , 		// Compare with the modbus feedback on equipement . 
		bReset		:= TON_CheckCommand[3].Q,
		bImpulsion	:= TRUE , 
		T			:= T#5S ) ;	
	
	// Autorization couplage 
	TON_CheckCommand[4](IN:= CheckCommand[4].bWarning , PT:= T#2S ) ; 
	CheckCommand[4](
		bCmd		:= MesDataExd.MesData.OUT_CmdAutCpl ,
		bMes		:= A1_SUBMV.MesDataExd.MesData.MesClosed_ALOFeederMVCB AND A1_SUBMV.MesDataExd.MesData.MesClosed_ALOFeederMVCB , 		// Compare with the modbus feedback on equipement . 
		bReset		:= TON_CheckCommand[4].Q,
		bImpulsion	:= TRUE , 
		T			:= T#5S ) ;
		
		(*
	// Manual Mode 
	TON_CheckCommand[5](IN:= CheckCommand[5].bWarning , PT:= T#2S ) ; 
	CheckCommand[5](
		bCmd		:= MesDataExd.MesData.OUT_CmdModeManuel ,
		bMes		:= A1_PP.MesDataExd.MesData.CalManualMode , 		// Compare with the modbus feedback on equipement . 
		bReset		:=TON_CheckCommand[5].Q ,
		bImpulsion	:= TRUE , 
		T			:= T#1S ) ;	
		
		*)
END_METHOD

METHOD M_Execute
//////////////////
//  Method Calls 
/////////////////
VAR 
	// Method local variables (reinitialized at each cycle) 
	// EMULATOR

	
END_VAR
// READING AND WRITING CLOCK //

// PERMANENT CONDITIONS //
	M_CP() ; 
	
// METHODS CALLS //
	IF bInit THEN
		M_Init() ; 
		bInit:= FALSE ; 
	ELSIF CmdInit_G THEN 
		bInit:= TRUE ;
	END_IF

	M_IEC104(); 
	M_Evaluate() ; 
	
	////////////////////
	M_AlarmManagement();
END_METHOD

METHOD M_IEC104
//////////////////
//  Read Modbus Variable for PCS . 
/////////////////
VAR 
	// Method local variables (reinitialized at each cycle) 
	
	bTest: BOOL;
	KK: BYTE;
END_VAR
	
FB_IEC(
	IN_bEnable := TRUE , //MesCP_Read , 
	AODB := AODB , 
	memory := ADR(memory) , 
	IN_Local := MesDataIEC.OUT_MesLocal ) ;
END_METHOD

METHOD M_Init
VAR 


END_VAR

// Initialize autorization couplage to false
IF bBoot AND NOT A1_SUBMV.MesDataExd.MesData.MesState.1 THEN 
	MesDataExd.MesData.OUT_CmdAutCpl := FALSE ;  // A VOIR SI ON VEUT MEMORISER CET ETAT OU PAS AU DEMARRAGE. Le.MesDataExd.MesData.est persistent.
	bBoot := FALSE ;
END_IF


///// INITIALIZE ////CstIPIEC104
// SERVER 1
	(* Configure protocol parameter *)
	FB_IEC.protPara.iK 				:= 12;(* default = 12 *)
	FB_IEC.protPara.iW 				:= 8;(* default = 8 *)
	FB_IEC.protPara.bThrottleMode 	:= TRUE;

	(* Configure system parameter *)
	FB_IEC.sysPara.asduAddr 		:= 1;
	FB_IEC.sysPara.bUsePCTime 		:= TRUE;
	FB_IEC.sysPara.bSyncTime 		:= TRUE;
	FB_IEC.sysPara.bSyncPCTime 		:= FALSE;
	FB_IEC.sysPara.bEndOfInit 		:= TRUE;
	FB_IEC.sysPara.bPerCyclic		:= TRUE;
	FB_IEC.sysPara.tPerCyclicBase	:= T#3S;
	FB_IEC.sysPara.bBackScan		:= FALSE;
	FB_IEC.sysPara.tBackScanCycle	:= T#3S;
	FB_IEC.sysPara.bPerFRZ			:= TRUE;
	FB_IEC.sysPara.tPerFRZCycle		:= T#15S;
	FB_IEC.sysPara.dbgMode 			:= (*IEC870_DEBUGMODE_ASDU OR*) IEC870_DEBUGMODE_DEVSTATE;

	(* Configure akuo iec104 parameter *)
	FB_IEC.akuoPara.iAOnb			:= 33 ; 
	FB_IEC.akuoPara.sLocalHost		:= CstIPIEC104 ; 
	
	initError := F_iecInitAOEntry( M_SP_TB_1, 12, IEC870_GRP_INROGEN, 0,  MAP_AREA_MEMORY, 10, 0, AODB[0] );		//OUT_MesLocal		       
	initError := F_iecInitAOEntry( M_SP_TB_1, 13, IEC870_GRP_INROGEN, 0,  MAP_AREA_MEMORY, 10, 1, AODB[1] );		//OUT_MesModeManuel_on
	initError := F_iecInitAOEntry( M_SP_TB_1, 14, IEC870_GRP_INROGEN, 0,  MAP_AREA_MEMORY, 10, 2, AODB[2] );      //OUT_MesModeAuto_on	 
	initError := F_iecInitAOEntry( M_SP_TB_1, 15, IEC870_GRP_INROGEN, 0,  MAP_AREA_MEMORY, 10, 3, AODB[3] );	    //OUT_MesCharging		   
	initError := F_iecInitAOEntry( M_SP_TB_1, 16, IEC870_GRP_INROGEN, 0,  MAP_AREA_MEMORY, 10, 4, AODB[4] );	    //OUT_MesDischarging	 
	initError := F_iecInitAOEntry( M_SP_TB_1, 20, IEC870_GRP_INROGEN, 0,  MAP_AREA_MEMORY, 10, 5, AODB[5] );      //OUT_MesEs			        
	initError := F_iecInitAOEntry( M_SP_TB_1, 21, IEC870_GRP_INROGEN, 0,  MAP_AREA_MEMORY, 10, 6, AODB[6] );	    //OUT_MesToS			       
	initError := F_iecInitAOEntry( M_SP_TB_1, 19, IEC870_GRP_INROGEN, 0,  MAP_AREA_MEMORY, 10, 7, AODB[7] );	    //OUT_MesIncident			   
	initError := F_iecInitAOEntry( M_SP_TB_1, 37, IEC870_GRP_INROGEN, 0,  MAP_AREA_MEMORY, 11, 0, AODB[8] );	    //OUT_MesFaultTeleMes		
	initError := F_iecInitAOEntry( M_SP_TB_1, 38, IEC870_GRP_INROGEN, 0,  MAP_AREA_MEMORY, 11, 1, AODB[9] );	    //OUT_MesFaultTeleCmd		
	initError := F_iecInitAOEntry( M_SP_TB_1, 39, IEC870_GRP_INROGEN, 0,  MAP_AREA_MEMORY, 11, 2, AODB[10] );	    //OUT_MesFaultTeleSgnl	
	initError := F_iecInitAOEntry( M_SP_TB_1, 41, IEC870_GRP_INROGEN, 0,  MAP_AREA_MEMORY, 11, 3, AODB[11] );	    //OUT_MesIECServerFault

		(* TSD *)
	initError := F_iecInitAOEntry( M_DP_TB_1, 43, IEC870_GRP_INROGEN, 0, MAP_AREA_MEMORY, 61, 2, AODB[12] );	//MesSoutirage_on			      	
	initError := F_iecInitAOEntry( M_DP_TB_1, 44, IEC870_GRP_INROGEN, 0, MAP_AREA_MEMORY, 61, 4, AODB[13] );   //MesComTest_on		     
	initError := F_iecInitAOEntry( M_DP_TB_1, 17, IEC870_GRP_INROGEN, 0, MAP_AREA_MEMORY, 12, 4, AODB[14] );   //MesCentrale_Cpl		   
	initError := F_iecInitAOEntry( M_DP_TB_1, 22, IEC870_GRP_INROGEN, 0, MAP_AREA_MEMORY, 12, 6, AODB[15] );	//MesCentrale_indispo	
	initError := F_iecInitAOEntry( M_DP_TB_1, 51, IEC870_GRP_INROGEN, 0, MAP_AREA_MEMORY, 12, 0, AODB[33] );   //MesDJOpen		   


	
	(* Measured value , short floating point value *)
	initError := F_iecInitAOEntry( M_ME_NC_1, 5, IEC870_GRP_INROGEN OR IEC870_GRP_PERCYC , 1, MAP_AREA_MEMORY, 42, 0, AODB[16] );	// OUT_MesSoC 			    
	initError := F_iecInitAOEntry( M_ME_NC_1, 6, IEC870_GRP_INROGEN OR IEC870_GRP_PERCYC , 1, MAP_AREA_MEMORY, 14, 0, AODB[17] );  // OUT_MesSoH 			    
	initError := F_iecInitAOEntry( M_ME_NC_1, 1, IEC870_GRP_INROGEN OR IEC870_GRP_PERCYC , 1, MAP_AREA_MEMORY, 18, 0, AODB[18] );  // OUT_MesP 			      
	initError := F_iecInitAOEntry( M_ME_NC_1, 2, IEC870_GRP_INROGEN OR IEC870_GRP_PERCYC , 1, MAP_AREA_MEMORY, 22, 0, AODB[19] );  // OUT_MesQ 			      
	initError := F_iecInitAOEntry( M_ME_NC_1, 3, IEC870_GRP_INROGEN OR IEC870_GRP_PERCYC , 1, MAP_AREA_MEMORY, 26, 0, AODB[20] );  // OUT_MesU_HTA 		   
	initError := F_iecInitAOEntry( M_ME_NC_1, 4, IEC870_GRP_INROGEN OR IEC870_GRP_PERCYC , 1, MAP_AREA_MEMORY, 30, 0, AODB[21] );	// OUT_MesFreq 		    
	initError := F_iecInitAOEntry( M_ME_NC_1, 7, IEC870_GRP_INROGEN OR IEC870_GRP_PERCYC , 1, MAP_AREA_MEMORY, 34, 0, AODB[22] );  // OUT_MesPdispo_inj 
	initError := F_iecInitAOEntry( M_ME_NC_1, 8, IEC870_GRP_INROGEN OR IEC870_GRP_PERCYC , 1, MAP_AREA_MEMORY, 38, 0, AODB[23] );  // OUT_MesPdispo_abs 

	(* Single commands *)
	initError := F_iecInitAOEntry( C_SC_TA_1, 30, 0, 0, MAP_AREA_MEMORY, 60, 0, AODB[24] );	//	IN_CmdModeManuel
	initError := F_iecInitAOEntry( C_SC_TA_1, 31, 0, 0, MAP_AREA_MEMORY, 60, 1, AODB[27] );	//	IN_CmdModeManuelOff
	initError := F_iecInitAOEntry( C_SC_TA_1, 32, 0, 0, MAP_AREA_MEMORY, 60, 2, AODB[25] );   //  IN_CmdAut_Cpl	  
	initError := F_iecInitAOEntry( C_SC_TA_1, 33, 0, 0, MAP_AREA_MEMORY, 60, 3, AODB[26] );	//	CmdDisconnect	
	
	(* Double commands *)
	initError := F_iecInitAOEntry( C_DC_TA_1, 26, 0, 0, MAP_AREA_MEMORY, 61, 2, AODB[28] );	//  CmdSoutirage		    
	initError := F_iecInitAOEntry( C_DC_TA_1, 27, 0, 0, MAP_AREA_MEMORY, 61, 4, AODB[29] );	//  CmdTest			    

	(* Set point,  short floating point values *)
	initError := F_iecInitAOEntry( C_SE_TC_1, 36, 0, 0, MAP_AREA_MEMORY, 72, 0, AODB[30] );		//IN_SetptP 		 
	initError := F_iecInitAOEntry( C_SE_TC_1, 34, 0, 0, MAP_AREA_MEMORY, 64, 0, AODB[31] );		//IN_ParamPmax 
	initError := F_iecInitAOEntry( C_SE_TC_1, 35, 0, 0, MAP_AREA_MEMORY, 68, 0, AODB[32] );		//IN_ParamPmin
END_METHOD

END_FUNCTION_BLOCK

// ---- 01_Equipement_Library/Inverter/FB_INV_Base.TcPOU
FUNCTION_BLOCK FB_INV_Base
//////////////////
// PV INverter. Base FB. 
//////////////////

VAR_INPUT PERSISTENT
	// Parameters of the Object (instance/model specific) 
		ParamTempoComAlarm				: TIME := T#30S ; 			(* (s) Config : Tempo to detect LOC Alarm*)
		ParamTimeOutCurtail     		: TIME := T#45S ;			(* (s) Config : Tempo to curtail power at set value before Timeout warning*)
		{attribute 'OPC.UA.DA' := '1'} 
		ParamClockReadTime 				: TIME := TIME#2S;	  		(* (s) Read Modbus Frequency *)
		{attribute 'OPC.UA.DA' := '1'} 
		ParamClockWriteTime 			: TIME := TIME#500MS; 	  	(* (ms) Write Modbus Frequency *)
 		ParamTimeout					: TIME := T#5S ;		  	(* (s) Timeout for modbus reading *)
		ParamPn							: REAL ;      				(* (kW)   Nominal Capacity *)
		ParamQn							: REAL ;      				(* (kVAr) Nominal reactive power *)
		ParamPdc						: REAL;						(* (kWc) Power Crête use for power repartition *)
END_VAR

VAR_INPUT
		IN_SetptPlimit					: REAL;						// (kW) [P,H] Dynamic active Power limit setpoint (curtailing)  
		IN_SetptPlimit_Local			: REAL;						// (kW) [P,H] Dynamic active Power limit setpoint (curtailing)  
		IN_SetptQ						: REAL; 					// (kVar) Dynamic reactive power setpoints 	
		IN_CmdStart						: BOOL;						// (NA) [P,H] External Start Command
		IN_CmdStop 						: BOOL; 					// (NA) [P,H] External Stop Command 
		IN_CmdStop_Local				: BOOL; 					// (NA) [P,H] External Stop Command, only for this inverter
		IN_CmdStart_Local				: BOOL;						// (NA) [P,H] External Start Command, only for this inverter	
		                                                    		
		IN_CmdToggleRead				: BOOL ;            		
		IN_CmdToggleWrite				: BOOL ;            		
		IN_CmdReset_L					: BOOL ;					// (NA) External Reset Command
END_VAR

VAR
	// M_ALARMMNGMT VARIABLES //
		TON_ComAlarm				: TON ; 				// Tempo before deteting loss of communication. 
	    TON_ComWarning				: TON ; 				// Tempo before detecting loss of communication.                                                	
                                     		    	
		MesWarningCom				: BOOL ; 				// (NA) [P,H]  True if bad communication

		CalModbusWriteAlarm         : BOOL ; 				// (NA) Modbus Write Alarm synthesis


	// M_READ VARIABLES//
//	MesDataExd		      	: INV ; 				// (NA) [P,H,B] INV  Data Structure 


	// M_CURTAIL VARIABLES //
		FB_CheckCommand1		  	: FB_CheckCommand ; 	// (NA) Functionnal Block to check if Curtail limit Writing Successful
		FB_CheckSetPt		  		: FB_CheckSetPt ; 		// (NA) Functionnal Block to check if Q setpoint Writing Successful

		R_TRIG_Curtail				: R_TRIG ;

		CalCompareWarningCurtail	: BOOL ; 				// (NA) Curtail failed alarm						
		CalCompareWarningQSetpt		: BOOL ; 				// (NA) Curtail failed alarm						

		WriteCmdP 			 		: BOOL;					// Modbus Write Rising Edge 
		WriteCmdQ 			 		: BOOL;					// Modbus Write Rising Edge 
	

	// M_STARTSTOP//            	
		Trig_Cmd_Read				: R_TRIG; 
		Trig_Cmd_Write				: R_TRIG;  

		
		RS_Cmd_Read					: RS ; 	
		RS_Cmd_Write				: RS ; 	       	
		Trig_Local_Start			: R_Trig;
		Trig_Local_Stop				: R_Trig;
		Trig_Start					: R_Trig;
		Trig_Stop					: R_Trig;	         
		RS_StartStop				: RS ; 					// (NA) Bistable Function for Start and Stop 
		RS_StartStop_Local			: RS;					// (NA) Bistable Function for Start and Stop local                        	
		                       
	// M_STATEMANAGER//
		MesState					: BYTE ; 				// (NA) Cal [P,H,B] Bit 0: OFF , Bit 2 : Feeding Slave 	

	// M_CP VARIABLES //	
	
	//M_EXECUTE VARIABLES //
		TP1								: TP ; 				// (NA) Tempo to define Modbus Reading Frequency 
		TP2 							: TP ; 				// (NA) Tempo to define Modbus Writing Frequency
		
		ClockRead		AT %Q*				: BOOL;			// (NA) Modbus reading Clock
		ClockWrite 		AT %Q*				: BOOL;			// (NA) Modbus writing Clock 	
		MesCP_Read					: BOOL := TRUE;	(* Read function enable *)
		MesCP_Write					: BOOL := FALSE;	(* Write function enable *)

	//M_Init 
		bInit 							: BOOL := TRUE ; // Init variable	
END_VAR

METHOD M_AlarmManagement
//////////////////
// Manages IntelliGen Alarms
/////////////////

VAR 
	// Method local variables (reinitialized at each cycle) 

END_VAR
END_METHOD

METHOD M_CP
//////////////////
//  Emulator
/////////////////

VAR 
	// Method local variables (reinitialized at each cycle) 
	
END_VAR
Trig_Cmd_Read(CLK:=IN_CmdToggleRead);
Trig_Cmd_Write(CLK:=IN_CmdToggleWrite);

IF Trig_Cmd_Read.Q THEN
	IN_CmdToggleRead := FALSE;
	MesCP_Read  := NOT MesCP_Read;
END_IF


IF Trig_Cmd_Write.Q THEN
	IN_CmdToggleWrite := FALSE;
	MesCP_Write := NOT MesCP_Write;
END_IF
END_METHOD

{attribute 'object_name' := 'M_Curtail'}
METHOD M_Curtail
//////////////////
// Write Curtail Command through modbus to PV inverters.  
//////////////////
VAR 
	// Method local variables (reinitialized at each cycle) 
	
	
END_VAR
IF IN_SetptPlimit	> IN_SetptPlimit_Local THEN
	IN_SetptPlimit := IN_SetptPlimit_Local;			// Local protection, can't take more than local setpoint
END_IF			
		

(*
// 	COMPARE CONSISTENCY	
	FB_CheckCommand1(
		T				:= ParamTimeOutCurtail ,
		bCmd			:= WriteCmdP, 
		bMes			:= MesDataExd.MesData.MesP < IN_SetptPlimit*1.05 , // 5% margin
		bImpulsion		:= TRUE , 
		bReset 			:= GVL_CFG.CmdClearFault_G, 
		bWarning 		=> CalCompareWarningCurtail); 
			
	FB_CheckSetPt(
			T					:= ParamTimeOutCurtail,
			Tolerance 			:= 5, 
			Range 				:= MesDataExd.MesData.ParamPn, 
			bTrigger 			:= WriteCmdQ , 
			bSetpt 				:= IN_SetptQlimit , 
			bMes 				:= MesDataExd.MesData.MesQ , 
			bReset				:= GVL_CFG.CmdClearFault_G  OR MesState <4 , 
			bWarning 			=> CalCompareWarningQSetpt);
			
			
			*)
END_METHOD

METHOD M_Execute
//////////////////
//  Method Calls 
/////////////////

VAR 
	// Method local variables (reinitialized at each cycle) 

END_VAR
// READING AND WRITING CLOCK //
	TP1(IN:=NOT TP1.Q , PT:= ParamClockReadTime);
	ClockRead 				:= TP1.Q;
	
	TP2(IN:=NOT TP2.Q , PT:= ParamClockWriteTime);
	ClockWrite 				:= TP2.Q;
	
// PERMANENT CONDITIONS //	
	M_CP() ; 
	
// METHODS CALLS//
	M_Read();

	M_StateManager() ; 
	M_StartStop() ; 
	M_Curtail();
	
	M_AlarmManagement();
END_METHOD

{attribute 'object_name' := 'M_Read'}
METHOD M_Read
//////////
// Read Method for SMA : Modbus reading
//////////
VAR
	// Method local variables (reinitialized at each cycle) 
	
END_VAR
END_METHOD

METHOD M_StartStop
//////////////////
// Start and Stop AMG
/////////////////
VAR 
	// Method local variables (reinitialized at each cycle) 

END_VAR
//IN_CmdStart := IN_CmdStart	AND NOT IN_CmdStop_Local; // Local Protection, can't switch on if i am switch off in local
END_METHOD

METHOD M_StateManager
//////////////////
// Detect which is the state of the inverter. IF loss of communication MesState =0 , the last inverter state is kept .  
/////////////////

VAR 
	// Method local variables (reinitialized at each cycle) 

	
END_VAR
END_METHOD

END_FUNCTION_BLOCK

// ---- 01_Equipement_Library/Inverter/FB_INV_Smartlogger.TcPOU
FUNCTION_BLOCK FB_INV_Smartlogger EXTENDS FB_INV_Base
//////////////////
// SmartLogger Huawei
//////////////////

VAR_INPUT PERSISTENT
	// Parameters of the Object (instance specific)
	{attribute 'OPC.UA.DA' := '1'}  
	ParamIpAddress		   : STRING 	:= '127.0.0.1'; (* (NA)Config: IP Adress of PV INverter*)
	{attribute 'OPC.UA.DA' := '1'} 
	ParamUnitID 			: BYTE  := 0; 			  	(* (NA)   Modbus Unit ID. *)
	ParamNbINV				: BYTE:=1 ; 				(* Number of inverters behind the smartlogger *)
	{attribute 'OPC.UA.DA' := '1'}              		
	ParamnTcpPort			: UINT := 502;				(* TCP port number *)
	ParamPnomINV			: REAL:=60; 				(* (kW) Nominal Power For one inverter *)
	ParamSLNum				: BYTE ; 					(* (NA) Config :Numerous of the ESS in the PP*)
	ParamID_PTR				: UINT;						(* (NA) ID of the PTR where Smartlogger is located*)
END_VAR

VAR_OUTPUT
	//Child objects
	
END_VAR

VAR

	// M_READ VARIABLES//
	MesDataExd	AT %Q*		: SL_Huawei;

//		FB_ModbusRead_I1          	: ARRAY[1..CstNbINVperPTR_G] OF  FB_ModbusRead ; 		// (NA) FB for Modbus Reading
		FB_ModbusRead_I2          	: FB_ModbusRead ; 										// (NA) FB for Modbus Reading
		FB_ModbusRead_I3          	: FB_ModbusRead ; 										// (NA) FB for Modbus Reading
			
//		MesBlock1_Temp 				: ARRAY[1..CstNbINVperPTR_G] OF ARRAY[0..24]  OF WORD; 	// (NA) Temporary Block with multiple modbus reading (Caution : Double Word variables)
//		MesBlock1_Temp 				: ARRAY[0..25*CstNbINVperPTR_G-1]  OF WORD; 			// (NA) Temporary Block with multiple modbus reading (Caution : Double Word variables)
		MesBlock2_Temp 				: ARRAY[0..56] OF WORD;									// (NA) Temporary Block with multiple modbus reading (Caution : Double Word variables)
		MesBlock3_Temp 				: ARRAY[0..14] OF WORD;									// (NA) Temporary Block with multiple modbus reading (Caution : Double Word variables)
                                                                                    		
		                                                                            		
//		MesModbusReadAlarm 		  	: ARRAY[1..CstNbINVperPTR_G] OF BOOL ; 					// (NA) Modbus Read Alarm for all modbus frames		
		MesModbusReadAlarm2 		: BOOL ; 												// (NA) Modbus Read Alarm for all modbus frames			
		MesModbusReadAlarm3 		: BOOL ; 												// (NA) Modbus Read Alarm for all modbus frames			

//		MesModbusAlarmCode			: ARRAY[1..CstNbINVperPTR_G] OF UDINT;					// (NA) Modbus Read Alarm Code
		MesModbusAlarmCode2			: UDINT;												// (NA) Modbus Read Alarm Code
		MesModbusAlarmCode3			: UDINT;												// (NA) Modbus Read Alarm Code

	
	// M_CURTAIL VARIABLES //
		FB_ModbusWrite_I2 		  	: FB_ModbusWrite ; 										// (NA) Functionnal Block for Writing Curtail limit through modbus
		FB_ModbusWrite_I3 		  	: FB_ModbusWrite ; 										// (NA) Functionnal Block for Writing Curtail limit through modbus	
		MesModbusWriteCode          : UDINT ; 												// (NA) Modbus Write Alarm Code 			 
		MesModbusWriteCode2         : UDINT ; 												// (NA) Modbus Write Alarm Code 
	                                                                           		
		MesModbusCurtailAlarm		: BOOL ;				   								// (NA) Modbus Write Curtail Alarm 
		MesModbusCurtailAlarm2		: BOOL ;				   								// (NA) Modbus Write Curtail Alarm 
		WriteBlock_Temp 	AT %Q*	: ARRAY[0..3] OF WORD;				 					// Temporary Block with multiple modbus writing	 
		
END_VAR

METHOD M_AlarmManagement
//////////////////
// Manages IntelliGen Alarms
/////////////////

VAR 
	// Method local variables (reinitialized at each cycle) 
	FB_AlarmCodeManager : FB_AlarmCodeManager ; 

	KK					: BYTE;		// For Loop 
	
	ComWarning			: BOOL;		// Aggregated Wcommunication warning
	ComAlarm			: BOOL;		// Aggregated communication Alarm
	ComINVWarning			: BOOL;		// Aggregated Wcommunication warning
	ComINVAlarm			: BOOL;		// Aggregated communication Alarm
	
	INVAlarm			: BOOL ; // At least one inverter has an alarm
END_VAR
//COMMUNICATION//
	CalModbusWriteAlarm := MesModbusCurtailAlarm ; 
	
	ComWarning 			:= MesModbusCurtailAlarm ;			// At least one modbus trame did not work
	ComAlarm			:= TRUE;						// All modbus trame did not work
	
		ComWarning 	:= ComWarning OR  MesModbusReadAlarm2 OR MesModbusReadAlarm3; // Smart logger LOC
		ComAlarm	:= ComAlarm  AND MesModbusReadAlarm2 AND MesModbusReadAlarm3; 
		
//		ComINVWarning := FALSE ; // LOC with inverters
//		ComINVAlarm	 := TRUE ; 
//		INVAlarm		:=FALSE ; 
		
(*	FOR KK:=1 TO ParamNbINV DO 
		ComINVWarning 	:= ComINVWarning OR MesDataExd.MesData.LExd.MesDataExd.MesData.NV[KK].CalComAlarm;
	    ComINVAlarm	:= ComINVAlarm  AND MesDataExd.MesData.LExd.MesDataExd.MesData.NV[KK].CalComAlarm ;
		INVAlarm := INVAlarm AND MesDataExd.MesData.LExd.MesDataExd.MesData.NV[KK].MesAlarm ;
	END_FOR
	*)	
	//Warning
	MesWarningCom 	:= ComWarning ;  
	//Alarm
	TON_ComAlarm(IN:= ComAlarm , PT:= ParamTempoComAlarm, Q=> MesDataExd.MesData.MesAlarmCom) ;	

// ALARM CODE //
	FB_AlarmCodeManager(
		bAlarm1			:= MesDataExd.MesData.MesState_Inv=6 ,	// Smart Logger general alarm (desactivate if LOC)  
		bAlarm2			:= MesDataExd.MesData.MesAlarmCom,  // Loss of communication with smart logger #COM
		bAlarm3			:=ComINVAlarm AND NOT MesWarningCom , 		// LOC with all inverters while they were connected
		bAlarm4			:=MesModbusCurtailAlarm, 		// 
		bAlarm5			:=FALSE, 
		bAlarm6			:=FALSE, 
		bAlarm7			:=FALSE, 
		bAlarm8			:=FALSE, 
		bAlarm9			:=FALSE, 
		bAlarm10		:=FALSE, 
		bAlarm11		:=FALSE, 
		bAlarm12		:=FALSE, 
		bAlarm13		:=FALSE, 
		bAlarm14		:=FALSE, 													// 
		bAlarm15		:= FALSE , 									// Command Alarm in case of intervention
		wAlarmCode		=>MesDataExd.MesData.MesAlarmCode);

// WARNING CODE //
	FB_AlarmCodeManager(
 		bAlarm1			:= ComINVWarning,								// At least one inverter has a loss of communication
		bAlarm2			:= CalCompareWarningCurtail,					// Measured Power above curtail Power 
		bAlarm3			:= MesWarningCom,								// Bad communication #COM
		bAlarm4			:=INVAlarm, 		// At least one inverter has an alarm
		bAlarm5			:=FALSE, 
		bAlarm6			:=FALSE, 
		bAlarm7			:=FALSE, 
		bAlarm8			:=FALSE, 
		bAlarm9			:=FALSE, 
		bAlarm10		:=FALSE, 
		bAlarm11		:=FALSE, 
		bAlarm12		:=FALSE, 
		bAlarm13		:=FALSE, 
		bAlarm14		:=FALSE, 
		bAlarm15		:=FALSE, 
		wAlarmCode		=>MesDataExd.MesData.MesWarningCode);	

// EVENT CODE //
	FB_AlarmCodeManager(
		bAlarm1			:= RS_StartStop.Q1, 			// Start command
		bAlarm2			:= NOT RS_StartStop.Q1, 		// Stop command
		bAlarm3			:= MesDataExd.MesData.MesState_Inv=2 OR MesDataExd.MesData.MesState_Inv=3, 		// Curtailing is ON
		bAlarm4			:= FALSE, 		// 
		bAlarm5			:= FALSE, 
		bAlarm6			:= FALSE, 
		bAlarm7			:= FALSE, 
		bAlarm8			:= FALSE, 
		bAlarm9			:= FALSE, 
		bAlarm10		:= FALSE, 
		bAlarm11		:= FALSE, 
		bAlarm12		:= FALSE, 
		bAlarm13		:= FALSE, 
		bAlarm14		:= FALSE, 
		bAlarm15		:= FALSE, 
		wAlarmCode		=>MesDataExd.MesData.MesEventCode);
END_METHOD

{attribute 'object_name' := 'M_Curtail'}
METHOD M_Curtail
//////////////////
// Write Curtail Command through modbus to PV inverters.  
//////////////////
VAR 
	// Method local variables (reinitialized at each cycle) 
	
	Threshold 			 : INT:=5 ;					// (0-100) Change percentage of Range to trigger the write commAND  

	CHECK				 : BOOL; 					// Check if changes. 
	WriteCmd 			 : BOOL;					// Modbus Write Rising Edge 
	
	SetptPlimit_Temp: ARRAY[0..1] OF WORD;
	SetptQlimit_Temp: ARRAY[0..1] OF WORD;
	
	WriteBlock_Temp1 				: ARRAY[0..1] OF WORD; 	// Temporary Block with multiple modbus writing	 
	WriteBlock_Temp2 				: ARRAY[0..1] OF WORD; 	// Temporary Block with multiple modbus writing	
	
	Split		: FB_SplitRealToWords ; 
	
	CHECK2: BOOL;

	CalInhibeWrite: BOOL;


	Quantity: BYTE;
END_VAR
// MODBUS VARIABLE FORMATING //
MesDataExd.MesData.OUT_SetptPLimit	:= MIN(MesDataExd.MesSetptPMax,MAX(0, IN_SetptPlimit)) ; 
MesDataExd.MesData.OUT_SetptQ	:= MIN(MesDataExd.MesSetptQMax , MAX(MesDataExd.MesSetptQMin , IN_SetptQ)) ; 
		
	
	Split(IN:= MesDataExd.MesData.OUT_SetptPLimit*10.0 , OUT=>SetptPlimit_Temp ) ;   //Between 0 and 100% Pmax
	Split(IN:= MesDataExd.MesData.OUT_SetptQ*10.0 , OUT=>SetptQlimit_Temp ) ; // Cosphi limité à 0.8
	
	
	WriteBlock_Temp1[0] := SetptPlimit_Temp[0] ; 
	WriteBlock_Temp1[1] := SetptPlimit_Temp[1] ; 
	WriteBlock_Temp2[0] := SetptQlimit_Temp[0] ; 
	WriteBlock_Temp2[1] := SetptQlimit_Temp[1] ; 

// MODBUS REQUEST //	
	// Modbus Blocks write
	FB_ModbusWrite_I2(
		pSrcAddr 			:= ADR(WriteBlock_Temp1) ,
		cbLength			:= SIZEOF(WriteBlock_Temp1) , 
		nQuantity 			:= 2,
		Reset				:= CmdClearFault_G, 
		sIPAddr				:=ParamIpAddress ,
		nTCPport			:= ParamnTcpPort ,  
		nUnitID				:=ParamUnitID , 
		nMBAddr				:=40424 , 
		tTimeout			:=ParamTimeout ,
		WriteCmd			:=ClockWrite AND MesCP_Write, 
		ModbusWriteAlarm	=>MesModbusCurtailAlarm , 
		ErrorId				=> MesModbusWriteCode); 

	FB_ModbusWrite_I3(
		pSrcAddr 			:= ADR(WriteBlock_Temp2) ,
		cbLength			:= SIZEOF(WriteBlock_Temp2) , 
		nQuantity 			:= 2,
		Reset				:= CmdClearFault_G, 
		sIPAddr				:=ParamIpAddress ,
		nTCPport			:= ParamnTcpPort ,  
		nUnitID				:=ParamUnitID , 
		nMBAddr				:=40426 , 
		tTimeout			:=ParamTimeout ,
		WriteCmd			:=ClockWrite AND MesCP_Write, 
		ModbusWriteAlarm	=>MesModbusCurtailAlarm2 , 
		ErrorId				=> MesModbusWriteCode2); 

	IF FB_ModbusWrite_I2.Completed THEN
		MesDataExd.OUT_SetptPlimit 	:= IN_SetptPlimit ;
		MesDataExd.OUT_SetptQlimit	:= IN_SetptQ;
	END_IF
END_METHOD

METHOD M_Init
VAR_INPUT
END_VAR

VAR

END_VAR
 MesDataExd.OUT_SetptPlimit := 9999999 ; // initialize to absurd value , to force a write of setpoint at startup . 
MesDataExd.OUT_SetptQlimit	:= 9999999 ; // initiali
END_METHOD

{attribute 'object_name' := 'M_Read'}
METHOD M_Read
//////////
// Read Method for SMA : Modbus reading
//////////
VAR
	// Method local variables (reinitialized at each cycle) 
	MW 					: FB_MergeWordsToDint; 
	KK					: BYTE;						 // Index to loop over modbus blocks. 	

END_VAR
IF	MesDataExd.MesData.MesCP_Read THEN	
	
	// Datalogger //
		//INITIALIZING MODBUS REQUESTS //
		FB_ModbusRead_I2(ClockRead:= ClockRead AND MesDataExd.MesData.MesCP_Read, Reset:= CmdClearFault_G ,sIPAddr:=ParamIpAddress , nUnitID:= ParamUnitID, tTimeout:= ParamTimeout,nTcpPort := ParamnTcpPort);
		FB_ModbusRead_I3(ClockRead:= ClockRead AND MesDataExd.MesData.MesCP_Read, Reset:= CmdClearFault_G ,sIPAddr:=ParamIpAddress , nUnitID:= ParamUnitID, tTimeout:= ParamTimeout,nTcpPort := ParamnTcpPort);
	
	// MODBUS REQUEST//
		FB_ModbusRead_I2(
			nQuantity		:= 57, 
			nMBAddr			:= 40521, 
			cbLength		:= SIZEOF(MesBlock2_Temp) , 
			pDestAddr		:= ADR(MesBlock2_Temp) , 
			ModbusReadAlarm	=>MesModbusReadAlarm2 , 
			ErrorId			=> MesModbusAlarmCode2);
			
		FB_ModbusRead_I3(
			nQuantity		:= 15, 
			nMBAddr			:= 40685, 
			cbLength		:= SIZEOF(MesBlock3_Temp) , 
			pDestAddr		:= ADR(MesBlock3_Temp) , 
			ModbusReadAlarm	=>MesModbusReadAlarm3 , 
			ErrorId			=> MesModbusAlarmCode3);		
			
	
	// MODBUS BLOCKS SEPARATION	
			MW(WORD_STRONG:= MesBlock2_Temp[0], WORD_WEAK := MesBlock2_Temp[1],SIGNED:=FALSE, FIX:=3 , SIZE:=2, VAR_OUT := MesDataExd.MesData.MesPdc);
	
			MW(WORD_STRONG:= MesBlock2_Temp[4], WORD_WEAK := MesBlock2_Temp[5],SIGNED:=TRUE, FIX:=3 , SIZE:=2, VAR_OUT := MesDataExd.MesData.MesP);
			MW(WORD_STRONG:= MesBlock2_Temp[11],SIGNED:=TRUE, FIX:=3 , SIZE:=1, VAR_OUT := MesDataExd.MesData.MesCosPhi);
	
			MW(WORD_STRONG:= MesBlock2_Temp[23], WORD_WEAK := MesBlock2_Temp[24],SIGNED:=TRUE, FIX:=3 , SIZE:=2, VAR_OUT := MesDataExd.MesData.MesQ);
			MW(WORD_STRONG:= MesBlock2_Temp[33], WORD_WEAK := MesBlock2_Temp[34],SIGNED:=TRUE, FIX:=1 , SIZE:=2, VAR_OUT := MesDataExd.MesData.MesIdc);
			MW(WORD_STRONG:= MesBlock2_Temp[39], WORD_WEAK := MesBlock2_Temp[40],SIGNED:=FALSE, FIX:=1 , SIZE:=2, VAR_OUT := MesDataExd.MesETot);
			MW(WORD_STRONG:= MesBlock2_Temp[41], WORD_WEAK := MesBlock2_Temp[42],SIGNED:=FALSE, FIX:=1 , SIZE:=2, VAR_OUT := MesDataExd.MesEDay);
		MesDataExd.MesData.MesState_Inv:= MesBlock2_Temp[45];
			
			MW(WORD_STRONG:= MesBlock2_Temp[51],SIGNED:=TRUE, FIX:=0 , SIZE:=1, VAR_OUT := MesDataExd.MesI1);
			MW(WORD_STRONG:= MesBlock2_Temp[52],SIGNED:=TRUE, FIX:=0 , SIZE:=1, VAR_OUT := MesDataExd.MesI2);
			MW(WORD_STRONG:= MesBlock2_Temp[53],SIGNED:=TRUE, FIX:=0 , SIZE:=1, VAR_OUT := MesDataExd.MesI3);
			MW(WORD_STRONG:= MesBlock2_Temp[54],SIGNED:=FALSE, FIX:=1 , SIZE:=1, VAR_OUT := MesDataExd.MesU12);
			MW(WORD_STRONG:= MesBlock2_Temp[55],SIGNED:=FALSE, FIX:=1 , SIZE:=1, VAR_OUT := MesDataExd.MesU23);
			MW(WORD_STRONG:= MesBlock2_Temp[56],SIGNED:=FALSE, FIX:=1 , SIZE:=1, VAR_OUT := MesDataExd.MesU31);
		
		MW(WORD_STRONG:= MesBlock2_Temp[51],SIGNED:=TRUE, FIX:=0 , SIZE:=1, VAR_OUT := MesDataExd.MesI1);
		MW(WORD_STRONG:= MesBlock2_Temp[52],SIGNED:=TRUE, FIX:=0 , SIZE:=1, VAR_OUT := MesDataExd.MesI2);
		MW(WORD_STRONG:= MesBlock2_Temp[53],SIGNED:=TRUE, FIX:=0 , SIZE:=1, VAR_OUT := MesDataExd.MesI3);
		MW(WORD_STRONG:= MesBlock2_Temp[54],SIGNED:=FALSE, FIX:=1 , SIZE:=1, VAR_OUT := MesDataExd.MesU12);
		MW(WORD_STRONG:= MesBlock2_Temp[55],SIGNED:=FALSE, FIX:=1 , SIZE:=1, VAR_OUT := MesDataExd.MesU23);
		MW(WORD_STRONG:= MesBlock2_Temp[56],SIGNED:=FALSE, FIX:=1 , SIZE:=1, VAR_OUT := MesDataExd.MesU31);
	
		// Block 3
		MW(WORD_STRONG:= MesBlock3_Temp[0], SIGNED:=FALSE, FIX:=2 , SIZE:=1, VAR_OUT := MesDataExd.MesEff);
		MW(WORD_STRONG:= MesBlock3_Temp[8],WORD_WEAK := MesBlock3_Temp[9], SIGNED:=FALSE, FIX:=2 , SIZE:=2, VAR_OUT := MesDataExd.MesSetptQMax);
		MW(WORD_STRONG:= MesBlock3_Temp[10],WORD_WEAK := MesBlock3_Temp[11], SIGNED:=TRUE, FIX:=2 , SIZE:=2, VAR_OUT := MesDataExd.MesSetptQMin);
		MW(WORD_STRONG:= MesBlock3_Temp[12],WORD_WEAK := MesBlock3_Temp[13], SIGNED:=FALSE, FIX:=2 , SIZE:=2, VAR_OUT := MesDataExd.MesSetptPMax);
	MesDataExd.MesOn	:= 	MesBlock3_Temp[14].0 ; 	
	


END_IF
	
// Properties update
	ParamPn := ParamPnomINV * ParamNbINV ;
END_METHOD

METHOD M_StartStop
//////////////////
// Start and Stop AMG
/////////////////
VAR 
	// Method local variables (reinitialized at each cycle) 

END_VAR
RS_StartStop(SET:= IN_CmdStart , RESET1:= IN_CmdStop) ; 

IF NOT RS_StartStop.Q1 THEN 
	IN_SetptPlimit:= 0 ; 	// When setpoint is equals to zero, the inverter stops. 
END_IF
END_METHOD

METHOD M_StateManager
//////////////////
// Detect which is the state of the inverter. IF loss of communication MesState =0 , the last inverter state is kept .  
/////////////////

VAR 
	// Method local variables (reinitialized at each cycle) 

	
END_VAR
MesState 			:= 0  ; 
 
IF MesDataExd.MesOn THEN
	// ON State
	MesState.2 		:= 1 ; 		// At least one inverter is feeding power to the grid . 
ELSE
	// OFF State  
	MesState.0 		:= 1 ; 
	
END_IF
END_METHOD

END_FUNCTION_BLOCK

// ---- 01_Equipement_Library/Inverter/FB_INV_Sun2000KtlMo.TcPOU
FUNCTION_BLOCK FB_INV_Sun2000KtlMo EXTENDS FB_INV_Base

VAR_INPUT PERSISTENT
	// Parameters of the Object (instance specific)
	{attribute 'OPC.UA.DA' := '1'}  
	ParamIPAddress	   : STRING := '127.0.0.1'; 	(* (NA)Config: IP Adress of PV INverter*)
	{attribute 'OPC.UA.DA' := '1'} 	
	ParamTcpPort		: UINT := 502;				(* (NA)Modbus TCP port*)
	{attribute 'OPC.UA.DA' := '1'} 
	ParamUnitID 		: BYTE  := 1; 	  			(* (NA)   SMA Modbus Unit ID. *)
	ParamID_INV			: BYTE ; 		        	(* (NA) Config :Numerous of the ESS in the PP*)
	ParamID_PTR			: BYTE ; 		        	(* (NA) Config :Numerous of the ESS in the PP*)

END_VAR

VAR_OUTPUT
	//Child objects

END_VAR

VAR
	//M_Acknowledge
		
	// M_ALARMMNGMT VARIABLES //
	MesAlarmCode1			: WORD ; 
	MesAlarmCode2			: WORD ; 
	
	// M_READ VARIABLES//
		Trig_Read					: R_TRIG;

		FB_ModbusRead_I2          	: FB_ModbusRead ; 									// (NA) FB for Modbus Reading
		FB_ModbusRead_I3          	: FB_ModbusRead ; 									// (NA) FB for Modbus Reading

		MesBlock_Temp 				: ARRAY[1..2] OF ARRAY [1..125] OF WORD ; 			// (NA) Temporary Block with multiple modbus reading (Caution : Double Word variables)

		AX_Busy						: ARRAY[1..2] OF BOOL;
		AX_Error					: ARRAY[1..2] OF BOOL;
		AX_ErrorID					: ARRAY[1..2] OF UDINT;

		MesDataExd				AT %Q*	: INV_Huawei ; 

	// M_CP

		
	// M_STATEMANAGER//
	
	//M_EXECUTE VARIABLES //
		TP_READ						: LTP; 		//Tempo de cadencement FB Modbus
		RTrig						: R_Trig; 	//Front montant sur TP_READ.Q
		ReadBusy					: BOOL;		//FB Modbus en busy

	//M_CURTAIL 
	
		// M_CURTAIL VARIABLES //
	
		FB_ModbusWrite1 		  	: FB_ModbusWrite; 					// (NA) Functionnal Block for Writing Curtail limit through modbus
		FB_ModbusWrite2 		  	: FB_ModbusWrite; 					// (NA) Functionnal Block for Writing Curtail limit through modbus
	
		MesWriteBlock_Temp			: WORD;												// (NA) Temporary Block with multiple modbus writing	 
	
		MesModbusCurtailAlarm		: BOOL ;				   							// (NA) Modbus Write Curtail Alarm 
		MesModbusWriteCode          : UDINT ; 											// (NA) Modbus Write Alarm Code 			 
		
		WriteBlock_Temp1 				: WORD; 	// Temporary Block with multiple modbus writing	
		WriteBlock_Temp2 				: WORD; 	// Temporary Block with multiple modbus writing

	
END_VAR

METHOD M_AlarmManagement
//////////////////
// Manages IntelliGen Alarms
/////////////////

VAR 
	// Method local variables (reinitialized at each cycle) 
	FB_AlarmCodeManager : FB_AlarmCodeManager ; 

	KK					: BYTE;		// For Loop 
	

	ComAlarm: BOOL;
END_VAR
//COMMUNICATION//
// CALC INVERT STAT ERREUR //

ComAlarm :=AX_Error[1] OR AX_Error[2] ; 
TON_ComAlarm(IN:= ComAlarm , PT:= ParamTempoComAlarm, Q=>MesDataExd.MesData.MesAlarmCom) ;	

// ALARM CODE //
	FB_AlarmCodeManager(
		bAlarm1			:= MesDataExd.MesAlm1.0,		// High String Voltage #Equipment
		bAlarm2			:= MesDataExd.MesAlm1.1,		// DC Arc Fault #Equipment
		bAlarm3			:= MesDataExd.MesAlm1.2,		// String Reversed #Equipment
		bAlarm4			:= MesDataExd.MesAlm1.5, 	//    AFCI Self-test Fault    #Equipment 
		bAlarm5			:= MesDataExd.MesAlm1.6,	// Short circuit between phase to PE #Equipment
		bAlarm6			:= MesDataExd.MesAlm1.7,	 //Power Grid Failure #Equipment
		bAlarm7			:= MesDataExd.MesAlm1.8,     //Grid Undervoltage #Equipment
		bAlarm8			:= MesDataExd.MesAlm1.9,     //Grid Overvoltag #Equipment
		bAlarm9			:= MesDataExd.MesAlm1.10,    //Unbalanced Grid Voltage #Equipment
		bAlarm10		:= MesDataExd.MesAlm1.11,    //Grid Overfrequency #Equipment
		bAlarm11		:= MesDataExd.MesAlm1.12,    //Grid Underfrequency #Equipment
		bAlarm12		:= MesDataExd.MesAlm1.13,    //Grid Frequency Instability #Equipment
		bAlarm13		:= MesDataExd.MesAlm1.14,    //Output Overcurrent #Equipment
		bAlarm14		:= MesDataExd.MesAlm1.15, 	 //	Large DC of Output current	 #Equipment								
		bAlarm15		:= FALSE,//
		wAlarmCode		=> MesDataExd.MesData.MesAlarmCode);

// WARNING CODE //
	FB_AlarmCodeManager(
 		bAlarm1			:= MesDataExd.MesAlm2.0,//Abnormal Leakage Current #Equipment
		bAlarm2			:= MesDataExd.MesAlm2.1,//Abnormal Ground. #Equipment
		bAlarm3			:= MesDataExd.MesAlm2.2,//Low Insulation Res #Equipment
		bAlarm4			:= MesDataExd.MesAlm2.3,//High Temperature #Equipment
		bAlarm5			:= MesDataExd.MesAlm2.4,//Abnormal Equipment #Equipment
		bAlarm6			:= MesDataExd.MesAlm3.2,//High String Voltage to Ground #Equipment
		bAlarm7			:= MesDataExd.MesAlm2.5,//Upgrade Failed #Equipment
		bAlarm8			:= MesDataExd.MesAlm2.7,//Abnormal Monitor Unit #Equipment
		bAlarm9			:= MesDataExd.MesAlm3.1,//Built-in PID operation abnormal #Equipment
		bAlarm10		:= FALSE,//
		bAlarm11		:= FALSE,//
		bAlarm12		:= FALSE,//
		bAlarm13		:= FALSE,//
		bAlarm14		:= FALSE,//
		bAlarm15		:= MesDataExd.MesData.MesAlarmCom,//
		wAlarmCode		=> MesDataExd.MesData.MesWarningCode);	

// EVENT CODE //
	FB_AlarmCodeManager(
		bAlarm1			:= MesDataExd.MesAlm1.3, 			// PV String Backfeed #Equipment
		bAlarm2			:= MesDataExd.MesAlm1.4, 		// Abnormal String #Equipment
		bAlarm3			:= MesDataExd.MesAlm2.6,	// License Expired #Equipment
		bAlarm4			:= FALSE, 	
		bAlarm5			:= FALSE, 
		bAlarm6			:= FALSE, 
		bAlarm7			:= FALSE, 
		bAlarm8			:= FALSE, 
		bAlarm9			:= FALSE, 
		bAlarm10		:= FALSE, 
		bAlarm11		:= FALSE, 
		bAlarm12		:= FALSE, 
		bAlarm13		:= FALSE, 
		bAlarm14		:= FALSE, 
		bAlarm15		:= FALSE, 
		wAlarmCode		=> MesDataExd.MesData.MesEventCode);

(*

// ALARM CODE //
	FB_AlarmCodeManager(
		bAlarm0			:= , 	// standby
		bAlarm1			:= , 	// grid-connected
		bAlarm2			:= , 	// grid-connected normally
		bAlarm3			:= ,    // grid connection with derating due to power rationing
		bAlarm4			:= ,    // grid connection with derating due to internal causes of the solar inverter
		bAlarm5			:= ,    // normal stop
		bAlarm6			:= ,    // stop due to faults
		bAlarm7			:= ,    // stop due to power rationing
		bAlarm8			:= ,    // shutdown
		bAlarm9			:= ,    // spot check
		bAlarm10		:= ,    // 
		bAlarm11		:= ,    //
		bAlarm12		:= ,    //
		bAlarm13		:= ,    //
		bAlarm14		:= ,    //
		bAlarm15		:= ,	//
		wAlarmCode		=> MesDataExd.MesStateIndic);

// ALARM CODE //
	FB_AlarmCodeManager(
		bAlarm0			:= , 	// locking status (0: locked; 1: unlocked)
		bAlarm1			:= , 	// PV connection status (0: disconnected; 1: connected)
		bAlarm2			:= , 	// DSP data collection (0: no; 1: yes)
		bAlarm3			:= ,    // 
		bAlarm4			:= ,    // 
		bAlarm5			:= ,    // 
		bAlarm6			:= ,    // 
		bAlarm7			:= ,    // 
		bAlarm8			:= ,    // 
		bAlarm9			:= ,    // 
		bAlarm10		:= ,    // 
		bAlarm11		:= ,    //
		bAlarm12		:= ,    //
		bAlarm13		:= ,    //
		bAlarm14		:= ,    //
		bAlarm15		:= ,	//
		wAlarmCode		=> MesDataExd.MesOpeStatus);


*)
END_METHOD

METHOD M_CP
//////////////////
//  Emulator
/////////////////

VAR 
	// Method local variables (reinitialized at each cycle) 
	
END_VAR
SUPER^.M_CP() ; 

//CTU(CU:=ClockRead , RESET:=CTU.Q , PV:=14 ) ; 
 

MesCP_Read				:=MesCP_Read ;//AND ((CTU.CV MOD 4) = (ParamInvNum MOD 4))   ;
END_METHOD

{attribute 'object_name' := 'M_Curtail'}
METHOD M_Curtail
//////////////////
// Write Curtail Command through modbus to PV inverters.  
//////////////////
VAR 
	// Method local variables (reinitialized at each cycle) 
	SetptPlimit_Temp: INT;
	SetptQlimit_Temp: INT;	 
	
END_VAR

IF	MesDataExd.MesData.MesCP_Write THEN

// MODBUS VARIABLE FORMATING //
	MesDataExd.MesData.OUT_SetptPLimit	:= MIN(100,MAX(0, (IN_SetptPlimit/ParamPn)*100)) ; //Between 0 and 100% Pmax
	MesDataExd.MesData.OUT_SetptQ	:= MIN(1 , MAX(-1 , IN_SetptQ/ParamPn)) ; //Between -1 and 1
	
	SetptPlimit_Temp := REAL_TO_INT(MesDataExd.MesData.OUT_SetptPLimit*10);
	SetptQlimit_Temp := REAL_TO_INT(MesDataExd.MesData.OUT_SetptQ*1000);
	
	WriteBlock_Temp1 := INT_TO_WORD(SetptPlimit_Temp) ; 
	WriteBlock_Temp2 := INT_TO_WORD(SetptQlimit_Temp) ; 

	// MODBUS REQUEST //	
	// Modbus Blocks write
	
	FB_ModbusWrite1(
		pSrcAddr 			:= ADR(WriteBlock_Temp1), 
		cbLength			:= SIZEOF(WriteBlock_Temp1),
		nQuantity 			:= 1,
		Reset				:=CmdClearFault_G, 
		sIPAddr				:=ParamIPAddress ,
		nTCPport			:=ParamTcpPort ,  
		nUnitID				:=ParamUnitID , 
		nMBAddr				:=40125 , 
		tTimeout			:=ParamTimeout ,
		WriteCmd			:=ClockWrite AND MesDataExd.MesData.MesCP_Write, 
		ModbusWriteAlarm	=>MesModbusCurtailAlarm , 
		ErrorId				=> MesModbusWriteCode)
	; 
	
		FB_ModbusWrite2(
		pSrcAddr 			:= ADR(WriteBlock_Temp2), 
		cbLength			:= SIZEOF(WriteBlock_Temp2),
		nQuantity 			:= 1,
		Reset				:=CmdClearFault_G, 
		sIPAddr				:=ParamIPAddress ,
		nTCPport			:=ParamTcpPort ,  
		nUnitID				:=ParamUnitID , 
		nMBAddr				:=40123 , 
		tTimeout			:=ParamTimeout ,
		WriteCmd			:=ClockWrite AND MesDataExd.MesData.MesCP_Write, 
		ModbusWriteAlarm	=>MesModbusCurtailAlarm , 
		ErrorId				=> MesModbusWriteCode)
		
		
	; 

END_IF
END_METHOD

METHOD M_Init
VAR_INPUT
END_VAR

VAR

END_VAR
ParamPn := 60 ;

bInit := FALSE;
END_METHOD

{attribute 'object_name' := 'M_Read'}
METHOD M_Read
//////////
// Read Method for SMA : Modbus reading
//////////
VAR
	// Method local variables (reinitialized at each cycle) 
	KK					: BYTE;						 // Index to loop over modbus blocks. 	
	JJ					: BYTE;
	AX_Adr				: ARRAY[1..2] OF WORD 		:= [32000,	40120];
	AX_Qty				: ARRAY[1..2] OF WORD		:= [110,	100];
	AX_StructRTU		: ARRAY[1..2] OF Struct_InputRTU ;
	
	MW					: FB_MergeWordsToDint;
	MesModbusReadAlarm2: BOOL;
	MesModbusReadAlarm3: BOOL;
END_VAR


IF MesCP_Read THEN	

	//INITIALIZING MODBUS REQUESTS //
//FB_ModbusRead_I2.Param
FB_ModbusRead_I2(ClockRead:= ClockRead AND MesCP_Read, Reset:= CmdClearFault_G ,sIPAddr:=ParamIPAddress , nUnitID:= ParamUnitID, tTimeout:= ParamTimeout,nTcpPort := ParamTcpPort, ParamEnableRetryPause:= TRUE);
//FB_ModbusRead_I3(ClockRead:= ClockRead AND MesCP_Read, Reset:= CalFaultClear_G ,sIPAddr:=ParamIPAdress , nUnitID:= ParamUnitID, tTimeout:= ParamTimeout,nTcpPort := ParamnTcpPort);

// MODBUS REQUEST//
	FB_ModbusRead_I2(
		nQuantity		:= 110, 
		nMBAddr			:= 32000, 
		cbLength		:= SIZEOF(MesBlock_Temp[1]) , 
		pDestAddr		:= ADR(MesBlock_Temp[1]) , 
		ModbusReadAlarm	=>AX_Error[1] , 
		ErrorId			=> AX_ErrorID[1]);
(*		
	FB_ModbusRead_I3(
		nQuantity		:= 100, 
		nMBAddr			:= 40120, 
		cbLength		:= SIZEOF(MesBlock_Temp[2]) , 
		pDestAddr		:= ADR(MesBlock_Temp[2]) , 
		ModbusReadAlarm	=>AX_Error[2] , 
		ErrorId			=> AX_ErrorID[2]);		
*)		
	
// MODBUS BLOCKS SEPARATION	


MesDataExd.MesStateIndic := MesBlock_Temp[1][1];
MesDataExd.MesOpeStatus := MesBlock_Temp[1][3];
MesDataExd.MesAlm1 := MesBlock_Temp[1][9];
MesDataExd.MesAlm2 := MesBlock_Temp[1][10];
MesDataExd.MesAlm3 := MesBlock_Temp[1][11];

FOR KK:=1  TO 12 DO 
	MW(WORD_STRONG := MesBlock_Temp[1][17+(KK-1)*2], FIX := 1, SIGNED := TRUE, VAR_OUT := MesdataExd.STR[KK].MesUdc	);
	MW(WORD_STRONG := MesBlock_Temp[1][17+(KK-1)*2+1], FIX := 2, SIGNED := TRUE, VAR_OUT := MesdataExd.STR[KK].MesIdc	);
END_FOR

MW(WORD_STRONG := MesBlock_Temp[1][65],WORD_WEAK := MesBlock_Temp[1][66], FIX := 3, Size := 2, SIGNED := TRUE, VAR_OUT := MesdataExd.Mesdata.MesPdc);
MW(WORD_STRONG := MesBlock_Temp[1][67], FIX := 1, Size := 1, SIGNED := FALSE, VAR_OUT := MesdataExd.MesU12);
MW(WORD_STRONG := MesBlock_Temp[1][68], FIX := 1, Size := 1, SIGNED := FALSE, VAR_OUT := MesdataExd.MesU23);
MW(WORD_STRONG := MesBlock_Temp[1][69], FIX := 1, Size := 1, SIGNED := FALSE, VAR_OUT := MesdataExd.MesU31);
MW(WORD_STRONG := MesBlock_Temp[1][70], FIX := 1, Size := 1, SIGNED := FALSE, VAR_OUT := MesdataExd.MesV1);
MW(WORD_STRONG := MesBlock_Temp[1][71], FIX := 1, Size := 1, SIGNED := FALSE, VAR_OUT := MesdataExd.MesV2);
MW(WORD_STRONG := MesBlock_Temp[1][72], FIX := 1, Size := 1, SIGNED := FALSE, VAR_OUT := MesdataExd.MesV3);
MW(WORD_STRONG := MesBlock_Temp[1][73], WORD_WEAK := MesBlock_Temp[1][74], FIX := 3, Size := 2, SIGNED := TRUE, VAR_OUT := MesdataExd.MesI1);
MW(WORD_STRONG := MesBlock_Temp[1][75], WORD_WEAK := MesBlock_Temp[1][76], FIX := 3, Size := 2, SIGNED := TRUE, VAR_OUT := MesdataExd.MesI2);
MW(WORD_STRONG := MesBlock_Temp[1][77], WORD_WEAK := MesBlock_Temp[1][78], FIX := 3, Size := 2, SIGNED := TRUE, VAR_OUT := MesdataExd.MesI3);

MW(WORD_STRONG := MesBlock_Temp[1][81], WORD_WEAK := MesBlock_Temp[1][82], FIX := 3, Size := 2, SIGNED := FALSE, VAR_OUT := MesdataExd.Mesdata.MesP);
MW(WORD_STRONG := MesBlock_Temp[1][83], WORD_WEAK := MesBlock_Temp[1][84], FIX := 3, Size := 2, SIGNED := TRUE, VAR_OUT := MesdataExd.Mesdata.MesQ);
MW(WORD_STRONG := MesBlock_Temp[1][85], FIX := 3, Size := 1, SIGNED := 1, VAR_OUT := MesDataExd.Mesdata.MesCosPhi);
MW(WORD_STRONG := MesBlock_Temp[1][86], FIX := 2, Size := 1, SIGNED := 0, VAR_OUT := MesDataExd.Mesdata.MesFreq);
MW(WORD_STRONG := MesBlock_Temp[1][88], FIX := 1, Size := 1, SIGNED := 0, VAR_OUT := MesDataExd.Mesdata.MesTemp);
MW(WORD_STRONG := MesBlock_Temp[1][89], FIX := 3, Size := 1, SIGNED := 0, VAR_OUT := MesDataExd.Mesdata.MesInsuResistor);
MesdataExd.MesData.MesState_Inv:= MesBlock_Temp[1][90];

MW(WORD_STRONG := MesBlock_Temp[1][107], WORD_WEAK := MesBlock_Temp[1][108], FIX := 2, Size := 2, SIGNED := 0, VAR_OUT := MesdataExd.MesETot);
MW(WORD_STRONG := MesBlock_Temp[1][109], WORD_WEAK := MesBlock_Temp[1][110], FIX := 2, Size := 2, SIGNED := 0, VAR_OUT := MesdataExd.MesEDay);

END_IF

// Properties update.
MesDataExd.MesData.MesI := (MesDataExd.MesI1 + MesDataExd.MesI2 + MesDataExd.MesI3)/3;
MesDataExd.MesData.MesV := (MesDataExd.MesV1 + MesDataExd.MesV2 + MesDataExd.MesV3)/3;
MesDataExd.MesData.MesS := SQRT(MesDataExd.MesData.MesP*MesDataExd.MesData.MesP + MesDataExd.MesData.MesQ*MesDataExd.MesData.MesQ);

MesDataExd.MesData.MesCurtl := MesDataExd.MesData.MesState_Inv=16#0201 OR MesDataExd.MesData.MesState_Inv =16#0202 ; 
MesDataExd.MesData.ParamPn := ParamPn ;
END_METHOD

METHOD M_StateManager
//////////////////
// Detect which is the state of the inverter. IF loss of communication MesState =0 , the last inverter state is kept .  
/////////////////

VAR 
	// Method local variables (reinitialized at each cycle) 

	
END_VAR
 MesDataExd.MesData.MesIDState := 0;
 
IF (MesDataExd.MesData.MesState_Inv.0 OR MesDataExd.MesData.MesState_Inv.5 OR MesDataExd.MesData.MesState_Inv.6 OR MesDataExd.MesData.MesState_Inv.7 OR MesDataExd.MesData.MesState_Inv.8) THEN  // DO I Produce ? Or I am in normal state
	// OFF State  
	MesDataExd.MesData.MesIDState.0 		:= 1 ; 
	
ELSIF MesDataExd.MesData.MesState_Inv.1 OR MesDataExd.MesData.MesState_Inv.2 OR MesDataExd.MesData.MesState_Inv.3 OR MesDataExd.MesData.MesState_Inv.4 THEN
	// ON State
	MesDataExd.MesData.MesIDState.1 		:= 1 ;
	
END_IF

SUPER^.M_StateManager() ;
END_METHOD

END_FUNCTION_BLOCK

// ---- 01_Equipement_Library/IPC/FB_IPC.TcPOU
FUNCTION_BLOCK FB_IPC

VAR_INPUT PERSISTENT 
	ParamTempoRestart		: TIME 	:= T#30S ;	(*  (s)Tempo to wait before resupplying the IPC*)
	
END_VAR
      	
VAR_INPUT           	
	Heure_Local     		: TIMESTRUCT;
	IN_CmdRestart 			: BOOL;	
	IN_CmdReset_L			: BOOL;			// (NA) External Reset Command
	
END_VAR     

VAR_OUTPUT
	//Child objects
	OUT_CmdOpen_IO			: BOOL;	
END_VAR        	
      	
VAR                 	
	bInit					: BOOL := TRUE;	// Booleen d'initialisation
		
	TP_Restart				: TP;
	// State Mananger //
	MesState				: BYTE; 		// Cal  : state
	
	// M_Evaluate //	
	MesData			: IPC;
END_VAR

METHOD M_AlarmManagement
//////////////////
// Generates object alarms and manages resets. 
//////////////////

VAR 
	// Method local variables (reinitialized at each cycle) 
	FB_AlarmCodeManager		: FB_AlarmCodeManager ;  
END_VAR
	
// ALARM CODE //
	FB_AlarmCodeManager(
		bAlarm1				:= FALSE,						//
		bAlarm2				:= FALSE,                       //
		bAlarm3				:= FALSE,                       //
		bAlarm4				:= FALSE,                       //
		bAlarm5				:= FALSE,                       //
		bAlarm6				:= FALSE,                       //
		bAlarm7				:= FALSE,                       //
		bAlarm8				:= FALSE,                       //
		bAlarm9				:= FALSE,                       //
		bAlarm10			:= FALSE,                       //
		bAlarm11			:= FALSE,                       //
		bAlarm12			:= FALSE,						//
		bAlarm13			:= FALSE ,                      //
		bAlarm14			:= FALSE ,                      //
		bAlarm15			:= FALSE,                       //
		wAlarmCode			=>MesData.MesAlarmCode);       
			                                                
// WARNING CODE //                                          
	FB_AlarmCodeManager(
		bAlarm1				:= FALSE, 						//				
		bAlarm2				:= FALSE,                       //
		bAlarm3				:= FALSE,                       //
		bAlarm4				:= FALSE,                       //
		bAlarm5				:= FALSE,                       //
		bAlarm6				:= FALSE,                       //
		bAlarm7				:= FALSE,                       //
		bAlarm8				:= FALSE,                       //
		bAlarm9				:= FALSE,                       //
		bAlarm10			:= FALSE,                       //
		bAlarm11			:= FALSE,                       //
		bAlarm12			:= FALSE,                       //
		bAlarm13			:= FALSE,                       //
		bAlarm14			:= FALSE,                       //
		bAlarm15			:= FALSE,                       //
		wAlarmCode			=>MesData.MesWarningCode);
		
// EVENT CODE //
	FB_AlarmCodeManager(
		bAlarm1			:= OUT_CmdOpen_IO, 					// ADSL is running 
		bAlarm2			:= FALSE , 							//
		bAlarm3			:= FALSE,                           //
		bAlarm4			:= FALSE,                           //
		bAlarm5			:= FALSE,                           //
		bAlarm6			:= FALSE,                           //
		bAlarm7			:= FALSE,                           //
		bAlarm8			:= FALSE,                           //
		bAlarm9			:= FALSE,                           //
		bAlarm10		:= FALSE,                           //
		bAlarm11		:= FALSE,                           //
		bAlarm12		:= FALSE,                           //
		bAlarm13		:= FALSE,                           //
		bAlarm14		:= FALSE,                           //
		bAlarm15		:= FALSE,                           //
		wAlarmCode		=>MesData.MesEventCode);
END_METHOD

METHOD M_Execute : BOOL
VAR_INPUT
END_VAR
IF bInit THEN
	M_Init();
ELSIF CmdClearFault_G OR IN_CmdReset_L THEN
	bInit := TRUE;
ELSE
	M_OpenClose(); 
	M_StateManager();
END_IF
END_METHOD

METHOD M_Init : BOOL
VAR_INPUT
END_VAR
bInit := FALSE;
END_METHOD

METHOD M_OpenClose
//////////////////
// Manages restart of the IPC 
//////////////////

VAR 
	// Method local variables (reinitialized at each cycle) 
	
END_VAR

// Rest Command
TP_Restart(IN:= IN_CmdRestart , PT:=ParamTempoRestart) ;
OUT_CmdOpen_IO := TP_Restart.Q ;  // Impulsion that goes back to zero as soon as the state of the TP goes down 

IF  IN_CmdRestart THEN
	 IN_CmdRestart := FALSE;
END_IF
END_METHOD

METHOD M_StateManager
//////////////////
// IPC off -> State.2 = 1, IPC on -> State.0 = 1 
/////////////////

VAR 
	// Method local variables (reinitialized at each cycle) 
	
END_VAR
// OPERATIONNAL INDEX //
IF NOT  OUT_CmdOpen_IO THEN 
	MesState.2 := 1;
ELSE
	MesState.0 := 1;
END_IF
END_METHOD

END_FUNCTION_BLOCK

// ---- 01_Equipement_Library/Operation Meter/FB_PM_520x230.TcPOU
FUNCTION_BLOCK FB_PM_520x230 EXTENDS FB_PM_Base
//////////////////
// Measurement Solution based on Digiware, but access through PMS Socomec
//////////////////
VAR CONSTANT
	// Characteristics of the object (Same for all instances)
			
END_VAR

VAR_INPUT PERSISTENT
	// Parameters of the Object (instance specific) 
	{attribute 'OPC.UA.DA' := '1'} 
	ParamUnitID					: BYTE := 1 ;									// (NA)unit ID
	ParamInInterfaceSub			: BOOL := TRUE; 								// Serial interface RS422/RS485 TYPE (0:EL6021,1:SUB9)			
END_VAR

VAR_OUTPUT
	//Child objects
	
END_VAR
VAR
	//M_ALARMMANAGEMENT VARIABLES//
	                                                    								
                                                        								

	//M_READ VARIABLES//
		ModbusRTU					: FB_ModbusRTU;								// (NA) FB for Modbus Reading

		MesDataExd				: PM_Standard;								// (NA) Structure of the PM3250
		
		ObjectCom					: INT;										// (NA) Sequence index
									
		Busy						: BOOL;
		StepRead					: UINT;										// (NA) Step for reading 2 blocks of registers
		AX_TrigRead					: ARRAY[1..1] OF R_trig;
		MbStruct					: ARRAY[1..1] OF Struct_InputRTU;	
		MesBlock					: ARRAY[1..1] OF ARRAY[1..120] OF WORD;	
		AX_Addr						: ARRAY[1..1] OF UINT 	:= [19000];
		AX_Qty						: ARRAY[1..1] OF UINT	:= [86];
		AX_UnitId					: ARRAY[1..1] OF BYTE	:= [1];
		AX_Function					: ARRAY[1..1] OF UINT	:= [4];	
		AX_Priority					: ARRAY[1..1] OF UINT	:= [1];
		KK							: INT;
		ComError 					: BOOL;
	//M_INIT VARIABLES //
		OutFBCompleteted			: BOOL;
	// M_EXECUTE VARIABLES //
		
                              

 
END_VAR

METHOD M_AlarmManagement
//////////////////
// Digiware measurement tool alarm and warning management
/////////////////

VAR 
	// Method local variables (reinitialized at each cycle) 
	FB_AlarmCodeManager			: FB_AlarmCodeManager ; 
	
	KK							: BYTE ;		// For loop
	
	CMWarning					: BOOL;			// At least one Digiware device in Alarm
	CMAlarm						: BOOL;			// At least one Digiware device in Alarm
	
END_VAR
//ComError 	:= MbStruct[1].OutError^;
	
TON_ComAlarm(IN:= ComError , PT:= ParamTempoComAlarm, Q=>MesDataExd.MesData.MesAlarmCom) ;	
TON_ComWarning(IN:= ComError  , PT:= ParamTempoComAlarm, Q=>MesWarningCom) ;	

//					General com alarm : All the read FB fucked up


// ALARM CODE //
	FB_AlarmCodeManager(
		bAlarm1			:= MesDataExd.MesData.MesAlarmCom  , 					// Communication Alarm #COM
		bAlarm2			:=FALSE, 		// 
		bAlarm3			:=FALSE, 		// 
		bAlarm4			:=FALSE, 		// 
		bAlarm5			:=FALSE, //
		bAlarm6			:=FALSE, //
		bAlarm7			:=FALSE, //
		bAlarm8			:=FALSE, //
		bAlarm9			:=FALSE, //
		bAlarm10		:=FALSE, //
		bAlarm11		:=FALSE, //
		bAlarm12		:=FALSE, //
		bAlarm13		:=FALSE, //
		bAlarm14		:=FALSE, //
		bAlarm15		:= FALSE , 			// 			 
		wAlarmCode		=>MesDataExd.MesData.MesAlarmCode);

// WARNING CODE //
	FB_AlarmCodeManager(		
		bAlarm1			:=MesWarningCom	,				 // Communication Warning #COM
		bAlarm2			:=FALSE, 		// 
		bAlarm3			:=FALSE, 		// 
		bAlarm4			:=FALSE, 		// 
		bAlarm5			:=FALSE, //
		bAlarm6			:=FALSE, //
		bAlarm7			:=FALSE, //
		bAlarm8			:=FALSE, //
		bAlarm9			:=FALSE, //
		bAlarm10		:=FALSE, //
		bAlarm11		:=FALSE, //
		bAlarm12		:=FALSE, //
		bAlarm13		:=FALSE, //
		bAlarm14		:=FALSE, //
		bAlarm15		:=FALSE, //
		wAlarmCode		=>MesDataExd.MesData.MesWarningCode);		

// EVENT CODE //
END_METHOD

METHOD M_Evaluate : BOOL
VAR_INPUT
END_VAR
END_METHOD

METHOD M_Execute
//////////////////
//  Method Calls 
/////////////////
VAR 
	// Method local variables (reinitialized at each cycle) 
	// EMULATOR
		Psoltot		: REAL;		// Total Solar Power . 
		KK			: BYTE;		// For Loop
	
END_VAR
// READING AND WRITING CLOCK //
	TP1(IN:=NOT TP1.Q , PT:= ParamClockReadTime);
	ClockRead 		:= TP1.Q;

// PERMANENT CONDITIONS //
	MesCP_Read 					:= TRUE  ; 
	
// METHODS CALLS //
	IF bInit THEN
		M_Init() ; 
		bInit					:= FALSE ; 
		
	END_IF

	M_Read() ; 
	
// EMULATOR COM READ  /////////////
	
	
	////////////////////
	M_AlarmManagement();
END_METHOD

METHOD M_Init
VAR 

END_VAR
//Modbus RTU Relay
FOR KK := 1 TO 1 DO 
	MbStruct[KK].InBuffer 		:= ADR(MesBlock[KK]);
	MbStruct[KK].InFunction 	:= AX_Function[KK];
	MbStruct[KK].InQuantity 	:= AX_Qty[KK];
	MbStruct[KK].InStartAddr 	:= AX_Addr[KK];
	MbStruct[KK].InUnitID 		:= AX_UnitId[KK];
	
END_FOR
END_METHOD

METHOD M_Read
//////////////////
//  Read Modbus Variable for PCS . 
/////////////////
VAR 
	// Method local variables (reinitialized at each cycle) 
	MW 					: FB_MergeWordsToFloat; 
	KK					: BYTE;  						// FOR Loop 

	
END_VAR
// CP-Read / Write 

MesDataExd.MesData.MesCP_Read := MesCP_Read ; 
 

IF MesCP_Read  THEN	

ModbusRTU();


FOR KK := 1 TO 1 DO
	AX_TrigRead[KK](CLK  :=ClockRead) ; // CalLocalTimeStruct.wSecond MOD 5 = 0);
	IF AX_TrigRead[KK].Q THEN
		ModbusRTU.M_AddAction_FIFO(InStruct := MbStruct[KK], InPriority := AX_Priority[KK]);
	END_IF
	MbStruct[KK].OutError			:= ADR(ComError);
END_FOR  
						
// PROPERTIES UPDATE // 
	// Block 1
//MW( WORD_STRONG:= MesBlock_Temp[1][1], 	WORD_WEAK := MesBlock_Temp[1][2],	SIGNED:=TRUE, FIX:=0 , SIZE:=2, VAR_OUT := MesDataExd.MesData.MesI2);
	
MW( WORD_STRONG:= MesBlock[1][1], 	WORD_WEAK := MesBlock[1][2], 	VAR_OUT:= MesDataExd.MesData.MesV1);
MW( WORD_STRONG:= MesBlock[1][3], 	WORD_WEAK := MesBlock[1][4], 	VAR_OUT:= MesDataExd.MesData.MesV2);
MW( WORD_STRONG:= MesBlock[1][5], 	WORD_WEAK := MesBlock[1][6], 	VAR_OUT:= MesDataExd.MesData.MesV3);
MW( WORD_STRONG:= MesBlock[1][7], 	WORD_WEAK := MesBlock[1][8], 	VAR_OUT:= MesDataExd.MesData.MesU12);
MW( WORD_STRONG:= MesBlock[1][9], 	WORD_WEAK := MesBlock[1][10], VAR_OUT:= MesDataExd.MesData.MesU23);
                                                                                
MW( WORD_STRONG:= MesBlock[1][11], 	WORD_WEAK := MesBlock[1][12], VAR_OUT:= MesDataExd.MesData.MesU31);
MW( WORD_STRONG:= MesBlock[1][13], 	WORD_WEAK := MesBlock[1][14], VAR_OUT:= MesDataExd.MesData.MesI1);
MW( WORD_STRONG:= MesBlock[1][15], 	WORD_WEAK := MesBlock[1][16], VAR_OUT:= MesDataExd.MesData.MesI2);
MW( WORD_STRONG:= MesBlock[1][17], 	WORD_WEAK := MesBlock[1][18], VAR_OUT:= MesDataExd.MesData.MesI3);
MW( WORD_STRONG:= MesBlock[1][19], 	WORD_WEAK := MesBlock[1][20], VAR_OUT:= MesDataExd.MesData.MesIN);
MW( WORD_STRONG:= MesBlock[1][21], 	WORD_WEAK := MesBlock[1][22], VAR_OUT:= MesDataExd.MesData.MesP1);
MW( WORD_STRONG:= MesBlock[1][23], 	WORD_WEAK := MesBlock[1][24], VAR_OUT:= MesDataExd.MesData.MesP2);
MW( WORD_STRONG:= MesBlock[1][25], 	WORD_WEAK := MesBlock[1][26], VAR_OUT:= MesDataExd.MesData.MesP3);
                                                                                
MW( WORD_STRONG:= MesBlock[1][27], 	WORD_WEAK := MesBlock[1][28], VAR_OUT:= MesDataExd.MesData.MesP);
MW( WORD_STRONG:= MesBlock[1][35], 	WORD_WEAK := MesBlock[1][36], VAR_OUT:= MesDataExd.MesData.MesS);
MW( WORD_STRONG:= MesBlock[1][43], 	WORD_WEAK := MesBlock[1][44], VAR_OUT:= MesDataExd.MesData.MesQ);

//MW( WORD_STRONG_F:= MesBlock[1][7], 	WORD_WEAK_F := MesBlock[1][8], NUMBER_F= MesDataExd.MesData.MesP);
//MW( WORD_STRONG_F:= MesBlock[1][9], 	WORD_WEAK_F := MesBlock[1][10], NUMBER_F= MesDataExd.MesData.MesQ1);
//MW( WORD_STRONG_F:= MesBlock[1][11], 	WORD_WEAK_F := MesBlock[1][12], NUMBER_F= MesDataExd.MesData.MesQ2);
//MW( WORD_STRONG_F:= MesBlock[1][13], 	WORD_WEAK_F := MesBlock[1][14], NUMBER_F= MesDataExd.MesData.MesQ3);
//MW( WORD_STRONG_F:= MesBlock[1][15], 	WORD_WEAK_F := MesBlock[1][16], NUMBER_F= MesDataExd.MesData.MesQ);
//MW( WORD_STRONG_F:= MesBlock[1][23], 	WORD_WEAK_F := MesBlock[1][24], NUMBER_F= MesDataExd.MesData.MesS);

//MW( WORD_STRONG_F:= MesBlock_Temp[4][1], 	WORD_WEAK_F := MesBlock_Temp[4][2], NUMBER_F= MesDataExd.MesData.MesTanPhi);
//MW( WORD_STRONG_F:= MesBlock_Temp[4][3], 	WORD_WEAK_F := MesBlock_Temp[4][4], NUMBER_F= MesDataExd.MesData.MesFreq);
//
//MW( WORD_STRONG_F:= MesBlock_Temp[3][1], 	WORD_WEAK_F := MesBlock_Temp[3][2], NUMBER_F= MesDataExd.MesData.MesEActProd);
//MW( WORD_STRONG_F:= MesBlock_Temp[3][3], 	WORD_WEAK_F := MesBlock_Temp[3][4], NUMBER_F= MesDataExd.MesData.MesEActCons);
//MW( WORD_STRONG_F:= MesBlock_Temp[3][5], 	WORD_WEAK_F := MesBlock_Temp[3][6], NUMBER_F= MesDataExd.MesData.MesEReactProd);
//MW( WORD_STRONG_F:= MesBlock_Temp[3][7], 	WORD_WEAK_F := MesBlock_Temp[3][8], NUMBER_F= MesDataExd.MesData.MesEReactCons);
//MW( WORD_STRONG:= MesBlock_Temp[4][3], 	WORD_WEAK := MesBlock_Temp[4][4],	SIGNED:=TRUE, FIX:=0 , SIZE:=2, VAR_OUT := MesDataExd.MesData.MesFreq);
//MW( WORD_STRONG:= MesBlock_Temp[5][1], 	WORD_WEAK := MesBlock_Temp[5][2],	SIGNED:=TRUE, FIX:=0 , SIZE:=2, VAR_OUT := MesDataExd.MesData.MesEActProd);
//MW( WORD_STRONG:= MesBlock_Temp[5][3], 	WORD_WEAK := MesBlock_Temp[5][4],	SIGNED:=TRUE, FIX:=0 , SIZE:=2, VAR_OUT := MesDataExd.MesData.MesEActCons);
//MW( WORD_STRONG:= MesBlock_Temp[5][5], 	WORD_WEAK := MesBlock_Temp[5][6],	SIGNED:=TRUE, FIX:=0 , SIZE:=2, VAR_OUT := MesDataExd.MesData.MesEReactProd);
//MW( WORD_STRONG:= MesBlock_Temp[5][7], 	WORD_WEAK := MesBlock_Temp[5][8],	SIGNED:=TRUE, FIX:=0 , SIZE:=2, VAR_OUT := MesDataExd.MesData.MesEReactCons);
MesDataExd.Mesdata.MesP	:= MesDataExd.MesData.MesP / 1000.0;
MesDataExd.MesData.MesS	:= MesDataExd.MesData.MesS	/ 1000.0;
MesDataExd.MesData.MesP 	:= -1 * MesDataExd.MesData.MesP;
MesDataExd.MesData.MesP1 	:= -1 * MesDataExd.MesData.MesP1/ 1000.0;
MesDataExd.MesData.MesP2 	:= -1 * MesDataExd.MesData.MesP2/ 1000.0;
MesDataExd.MesData.MesP3 	:= -1 * MesDataExd.MesData.MesP3/ 1000.0;

MesDataExd.MesData.MesQ 	:= -1 * MesDataExd.MesData.MesQ;

MesDataExd.MesData.MesQ 	:= MesDataExd.MesData.MesQ/1000.0;

IF MesDataExd.MesData.MesP <> 0 THEN
MesDataExd.MesData.MesTanPhi := MesDataExd.MesData.MesQ /  MesDataExd.MesData.MesP;

ELSE
MesDataExd.MesData.MesTanPhi := 0;
END_IF



END_IF
END_METHOD

END_FUNCTION_BLOCK

// ---- 01_Equipement_Library/Operation Meter/FB_PM_Base.TcPOU
FUNCTION_BLOCK FB_PM_Base 
//////////////////
// Measurement Solution. Base FB
//////////////////
VAR_INPUT PERSISTENT
	// Parameters of the Object (instance specific) 
	ParamTempoComAlarm				: TIME 		:= T#10S ; 						(* (s) Config : Tempo to detect LOC Alarm*)
	{attribute 'OPC.UA.DA' := '1'} 
	ParamClockReadTime 				: TIME 		:= TIME#200MS;	  				(* (ms) Read Modbus period  *)
	ParamTimeout					: TIME  	:= T#2S ;			  			(* (s) Timeout for modbus reading*)
	
	
END_VAR

VAR_INPUT
	//Child objects
	IN_CmdToggleRead				: BOOL ; 
	IN_CmdReset_L					: BOOL ;									// (NA) External Reset Command

END_VAR
VAR
	//M_ALARMMANAGEMENT VARIABLES//
		TON_ComAlarm				: TON ; 									// Tempo before detecting loss of communication 
	    TON_ComWarning				: TON ; 									// Tempo before detecting loss of one frame                                               								
                                            								    
		MesWarningCom				: BOOL ; 									// True if bad communication 
                                                                                 
	//M_READ VARIABLES//                                                         
//	MesDataExd		AT %Q*	: PM ;                                 
		ClockRead			AT %Q*	: BOOL ;	 								// Clock Read
                                                                                
		                                                                         
	//M_INIT VARIABLES //
		bInit						: BOOL 				:= TRUE ; 							// (NA) Initialize object parameters at first cycle 
		                                                                         
	// M_EXECUTE VARIABLES //
		TP1							: TP ; 												// (NA) Tempo to define Modbus Reading Frequency  
                                                             	                                                                                                                                                      
		//MesCP_Read					: BOOL;													// (NA) Permanent conditions to activate method
        Trig_Cmd_Read				: R_TRIG;      

